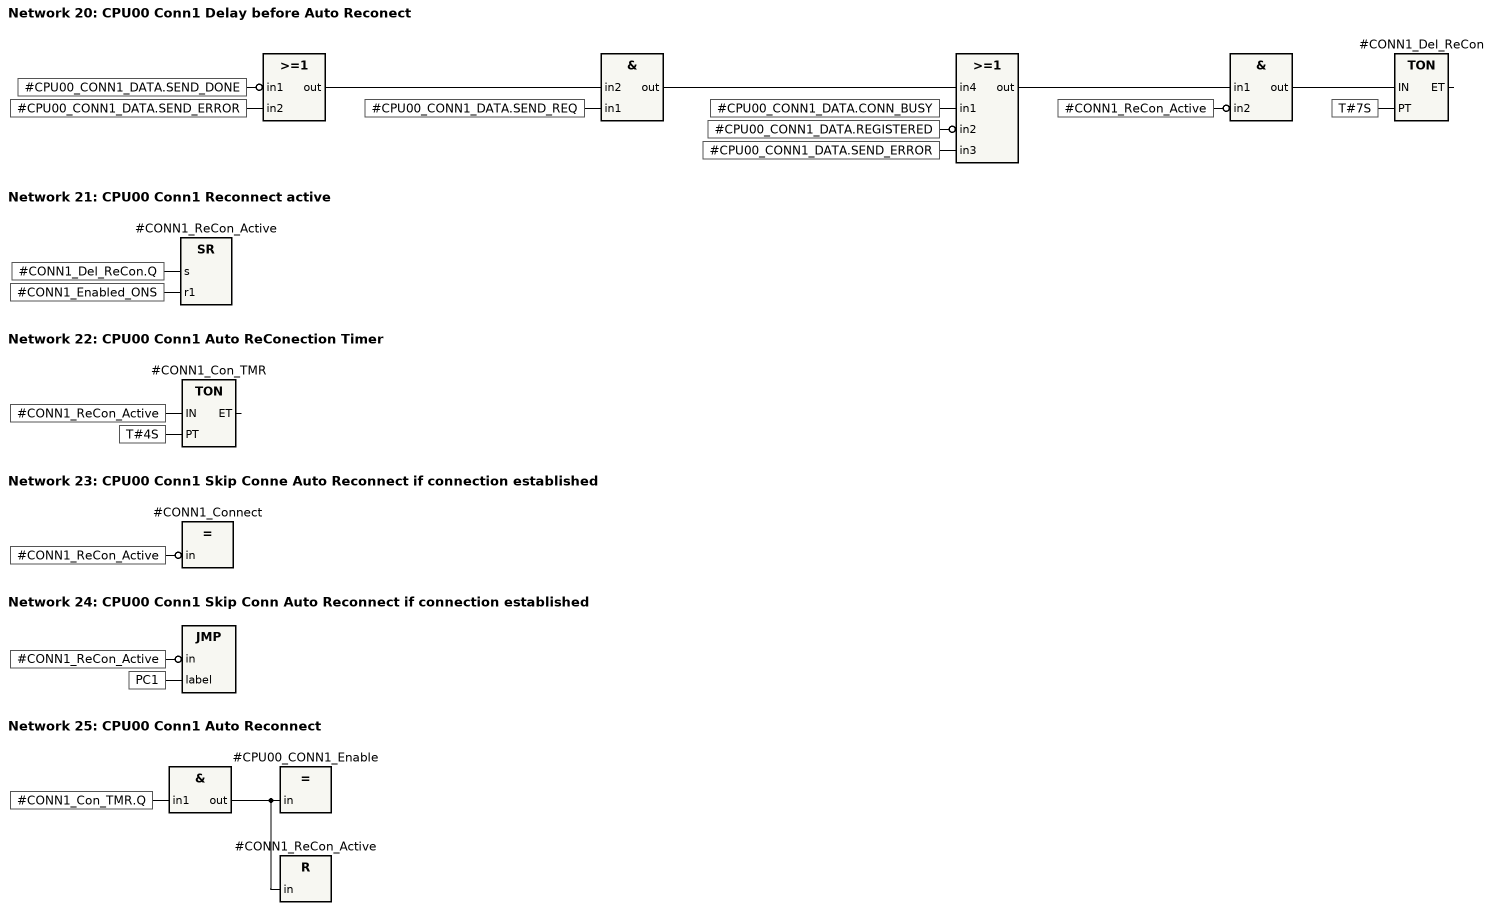
   #CONN1_Del_ReCon(IN := (((NOT #CPU00_CONN1_DATA.SEND_DONE OR #CPU00_CONN1_DATA.SEND_ERROR) AND #CPU00_CONN1_DATA.SEND_REQ) OR #CPU00_CONN1_DATA.CONN_BUSY OR NOT #CPU00_CONN1_DATA.REGISTERED OR #CPU00_CONN1_DATA.SEND_ERROR) AND NOT #CONN1_ReCon_Active,   // TON
                    PT := T#7S);
END_REGION

REGION Network 21: CPU00 Conn1 Reconnect active
   IF #CONN1_Del_ReCon.Q THEN
       #CONN1_ReCon_Active := TRUE;   // SR flip-flop
   END_IF;
   IF #CONN1_Enabled_ONS THEN #CONN1_ReCon_Active := FALSE; END_IF;
END_REGION

REGION Network 22: CPU00 Conn1 Auto ReConection Timer
   #CONN1_Con_TMR(IN := #CONN1_ReCon_Active, PT := T#4S);   // TON
END_REGION

REGION Network 23: CPU00 Conn1 Skip Conne Auto Reconnect if connection established
   #CONN1_Connect := NOT #CONN1_ReCon_Active;
END_REGION

REGION Network 24: CPU00 Conn1 Skip Conn Auto Reconnect if connection established
   IF NOT #CONN1_ReCon_Active THEN GOTO PC1; END_IF;
END_REGION

REGION Network 25: CPU00 Conn1 Auto Reconnect
   #CPU00_CONN1_Enable := #CONN1_Con_TMR.Q;
   IF #CONN1_Con_TMR.Q THEN #CONN1_ReCon_Active := FALSE; END_IF;
END_REGION

REGION Network 26 (STL): CPU00 Conn1 Set initial connection bit
   PC1:  O     #MASTER_LINK.FIRST_SCAN;
         O(;
         A     #CPU00_CONN1_Enable;
         FP    #CONN1_En_ONS;
         =     #CONN1_Enabled_ONS;
         A     #CONN1_Enabled_ONS;
         );
         =     #CONN1_INIT_COM;
END_REGION

REGION Network 27: CPU00 Conn1 Clear Bits to start initial conn and communication
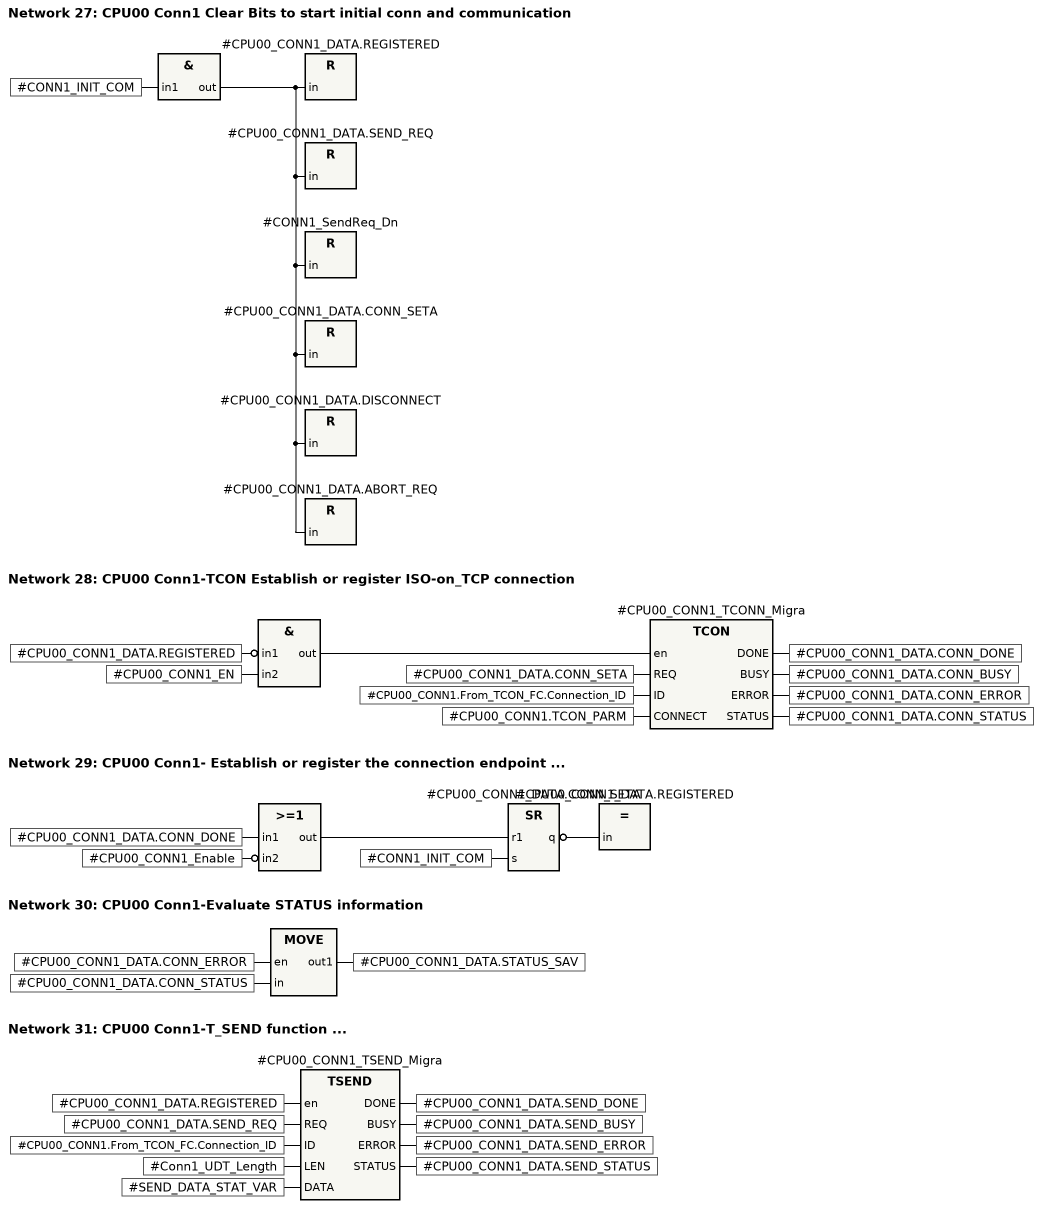
   IF #CONN1_INIT_COM THEN
       #CPU00_CONN1_DATA.REGISTERED := FALSE;
       #CPU00_CONN1_DATA.SEND_REQ := FALSE;
       #CONN1_SendReq_Dn := FALSE;
       #CPU00_CONN1_DATA.CONN_SETA := FALSE;
       #CPU00_CONN1_DATA.DISCONNECT := FALSE;
       #CPU00_CONN1_DATA.ABORT_REQ := FALSE;
   END_IF;
END_REGION

REGION Network 28: CPU00 Conn1-TCON Establish or register ISO-on_TCP connection
   // After the connection has been established, it is automatically monitored and 
   // maintained by the operating system of the CPU.
   // 
   // If the connection has been interrupted, by any line break or due to the remote 
   // communications partner, the active partner attempts to reestablish the 
   // connection.
   // 
   // Therefore, the FB 65 "TCON" may not be called again!
   IF NOT #CPU00_CONN1_DATA.REGISTERED AND #CPU00_CONN1_EN THEN
       #CPU00_CONN1_TCONN_Migra(REQ := #CPU00_CONN1_DATA.CONN_SETA,   // TCON
                               ID := #CPU00_CONN1.From_TCON_FC.Connection_ID,
                               CONNECT := #CPU00_CONN1.TCON_PARM,
                               DONE => #CPU00_CONN1_DATA.CONN_DONE,
                               BUSY => #CPU00_CONN1_DATA.CONN_BUSY,
                               ERROR => #CPU00_CONN1_DATA.CONN_ERROR,
                               STATUS => #CPU00_CONN1_DATA.CONN_STATUS);
   END_IF;
END_REGION

REGION Network 29: CPU00 Conn1- Establish or register the connection endpoint ...
   // while startup phase (initial).
   // 
   // Indication of the connection status:
   // 
   // a) If the CPU may establish the specified connection after Stop/Run  
   // immediately, the variable "REGISTERED" indicates HIGH (=1).
   // 
   // b) If the CPU is not able to establish the specified connection after Stop/Run, 
   // the variable "REGISTERED" remains LOW(=0).
   // 
   // c) Note: If the instance DB is loaded by the user, the variable "REGISTERED" 
   // indicates HIGH, although the connection may not be established yet. 
   // However, the FB64 "TRCV" would indicate the STATUS=0x80C4, as long as the 
   // connection has not been established.
   IF #CONN1_INIT_COM THEN
       #CPU00_CONN1_DATA.CONN_SETA := TRUE;   // SR flip-flop
   END_IF;
   IF #CPU00_CONN1_DATA.CONN_DONE OR NOT #CPU00_CONN1_Enable THEN
       #CPU00_CONN1_DATA.CONN_SETA := FALSE;
   END_IF;
   #CPU00_CONN1_DATA.REGISTERED := NOT #CPU00_CONN1_DATA.CONN_SETA;
END_REGION

REGION Network 30: CPU00 Conn1-Evaluate STATUS information
   // If ERROR occured then save STATUS!
   IF #CPU00_CONN1_DATA.CONN_ERROR THEN
       #CPU00_CONN1_DATA.STATUS_SAV := #CPU00_CONN1_DATA.CONN_STATUS;
   END_IF;
END_REGION

REGION Network 31: CPU00 Conn1-T_SEND function ...
   // if connection is established to transmit the data to the partner as a message.
   IF #CPU00_CONN1_DATA.REGISTERED THEN
       #CPU00_CONN1_TSEND_Migra(REQ := #CPU00_CONN1_DATA.SEND_REQ,   // TSEND
                               ID := #CPU00_CONN1.From_TCON_FC.Connection_ID,
                               LEN := #Conn1_UDT_Length,
                               DATA := #SEND_DATA_STAT_VAR,
                               DONE => #CPU00_CONN1_DATA.SEND_DONE,
                               BUSY => #CPU00_CONN1_DATA.SEND_BUSY,
                               ERROR => #CPU00_CONN1_DATA.SEND_ERROR,
                               STATUS => #CPU00_CONN1_DATA.SEND_STATUS);
   END_IF;
END_REGION

REGION Network 32: CPU00 Conn1-Generate the rising edge SEND_REQ to start T_SEND
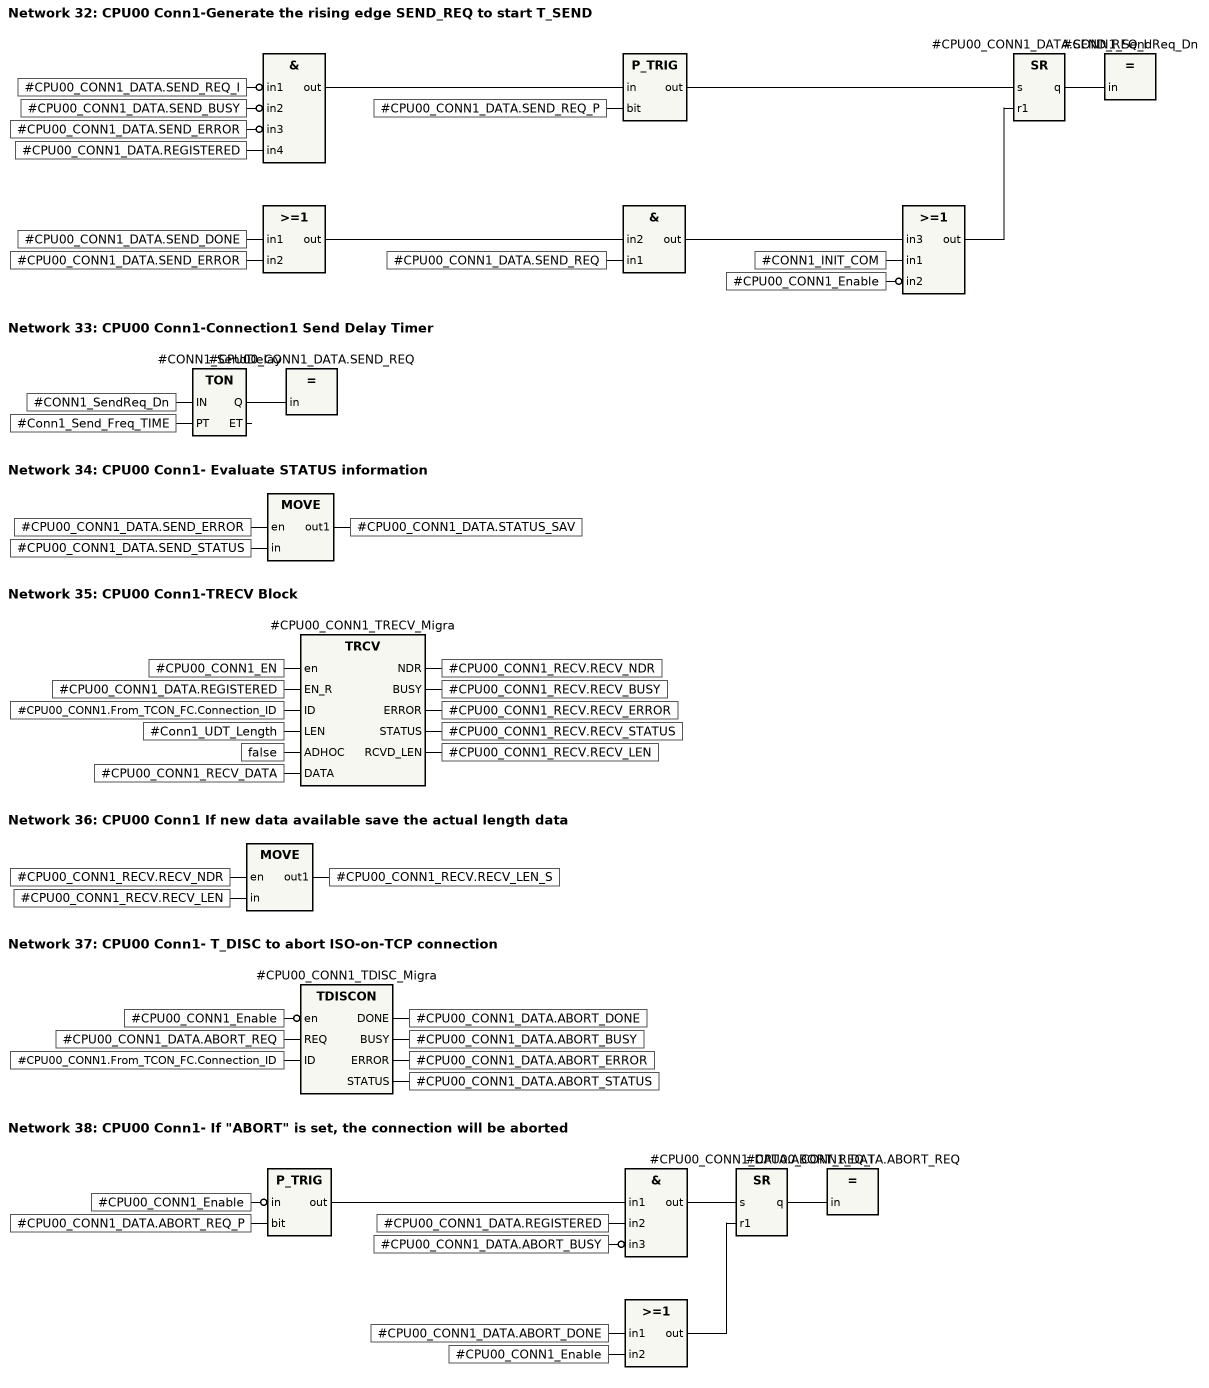
   #_w1 := NOT #CPU00_CONN1_DATA.SEND_REQ_I AND NOT #CPU00_CONN1_DATA.SEND_BUSY AND NOT #CPU00_CONN1_DATA.SEND_ERROR AND #CPU00_CONN1_DATA.REGISTERED;
   #_w2 := #_w1 AND NOT #CPU00_CONN1_DATA.SEND_REQ_P;   // rising edge
   #CPU00_CONN1_DATA.SEND_REQ_P := #_w1;
   IF #_w2 THEN
       #CPU00_CONN1_DATA.SEND_REQ_I := TRUE;   // SR flip-flop
   END_IF;
   IF ((#CPU00_CONN1_DATA.SEND_DONE OR #CPU00_CONN1_DATA.SEND_ERROR) AND #CPU00_CONN1_DATA.SEND_REQ) OR #CONN1_INIT_COM OR NOT #CPU00_CONN1_Enable THEN
       #CPU00_CONN1_DATA.SEND_REQ_I := FALSE;
   END_IF;
   #CONN1_SendReq_Dn := #CPU00_CONN1_DATA.SEND_REQ_I;
END_REGION

REGION Network 33: CPU00 Conn1-Connection1 Send Delay Timer
   #CONN1_SendDelay(IN := #CONN1_SendReq_Dn, PT := #Conn1_Send_Freq_TIME);   // TON
   #CPU00_CONN1_DATA.SEND_REQ := #CONN1_SendDelay.Q;
END_REGION

REGION Network 34: CPU00 Conn1- Evaluate STATUS information
   // If ERROR occured then save STATUS!
   IF #CPU00_CONN1_DATA.SEND_ERROR THEN
       #CPU00_CONN1_DATA.STATUS_SAV := #CPU00_CONN1_DATA.SEND_STATUS;
   END_IF;
END_REGION

REGION Network 35: CPU00 Conn1-TRECV Block
   IF #CPU00_CONN1_EN THEN
       #CPU00_CONN1_TRECV_Migra(EN_R := #CPU00_CONN1_DATA.REGISTERED,   // TRCV
                               ID := #CPU00_CONN1.From_TCON_FC.Connection_ID,
                               LEN := #Conn1_UDT_Length,
                               ADHOC := false,
                               DATA := #CPU00_CONN1_RECV_DATA,
                               NDR => #CPU00_CONN1_RECV.RECV_NDR,
                               BUSY => #CPU00_CONN1_RECV.RECV_BUSY,
                               ERROR => #CPU00_CONN1_RECV.RECV_ERROR,
                               STATUS => #CPU00_CONN1_RECV.RECV_STATUS,
                               RCVD_LEN => #CPU00_CONN1_RECV.RECV_LEN);
   END_IF;
END_REGION

REGION Network 36: CPU00 Conn1 If new data available save the actual length data
   IF #CPU00_CONN1_RECV.RECV_NDR THEN #CPU00_CONN1_RECV.RECV_LEN_S := #CPU00_CONN1_RECV.RECV_LEN; END_IF;
END_REGION

REGION Network 37: CPU00 Conn1- T_DISC to abort ISO-on-TCP connection
   // The FB 66 "TDISCON" terminates a communications connection from the CPU to a
   // communications partner.
   // 
   // An existing connection is terminated when FB 66 "TDISCON" is called or when the
   // CPU has gone into STOP mode. To reestablish the connection, the FB 65 "TCON" 
   // has to be invoked again.
   IF NOT #CPU00_CONN1_Enable THEN
       #CPU00_CONN1_TDISC_Migra(REQ := #CPU00_CONN1_DATA.ABORT_REQ,   // TDISCON
                               ID := #CPU00_CONN1.From_TCON_FC.Connection_ID,
                               DONE => #CPU00_CONN1_DATA.ABORT_DONE,
                               BUSY => #CPU00_CONN1_DATA.ABORT_BUSY,
                               ERROR => #CPU00_CONN1_DATA.ABORT_ERROR,
                               STATUS => #CPU00_CONN1_DATA.ABORT_STATUS);
   END_IF;
END_REGION

REGION Network 38: CPU00 Conn1- If "ABORT" is set, the connection will be aborted
   #_w1 := NOT #CPU00_CONN1_Enable AND NOT #CPU00_CONN1_DATA.ABORT_REQ_P;   // rising edge
   #CPU00_CONN1_DATA.ABORT_REQ_P := NOT #CPU00_CONN1_Enable;
   IF #_w1 AND #CPU00_CONN1_DATA.REGISTERED AND NOT #CPU00_CONN1_DATA.ABORT_BUSY THEN
       #CPU00_CONN1_DATA.ABORT_REQ_I := TRUE;   // SR flip-flop
   END_IF;
   IF #CPU00_CONN1_DATA.ABORT_DONE OR #CPU00_CONN1_Enable THEN
       #CPU00_CONN1_DATA.ABORT_REQ_I := FALSE;
   END_IF;
   #CPU00_CONN1_DATA.ABORT_REQ := #CPU00_CONN1_DATA.ABORT_REQ_I;
END_REGION

REGION Network 39: CPU00 Conn1-Communication OK
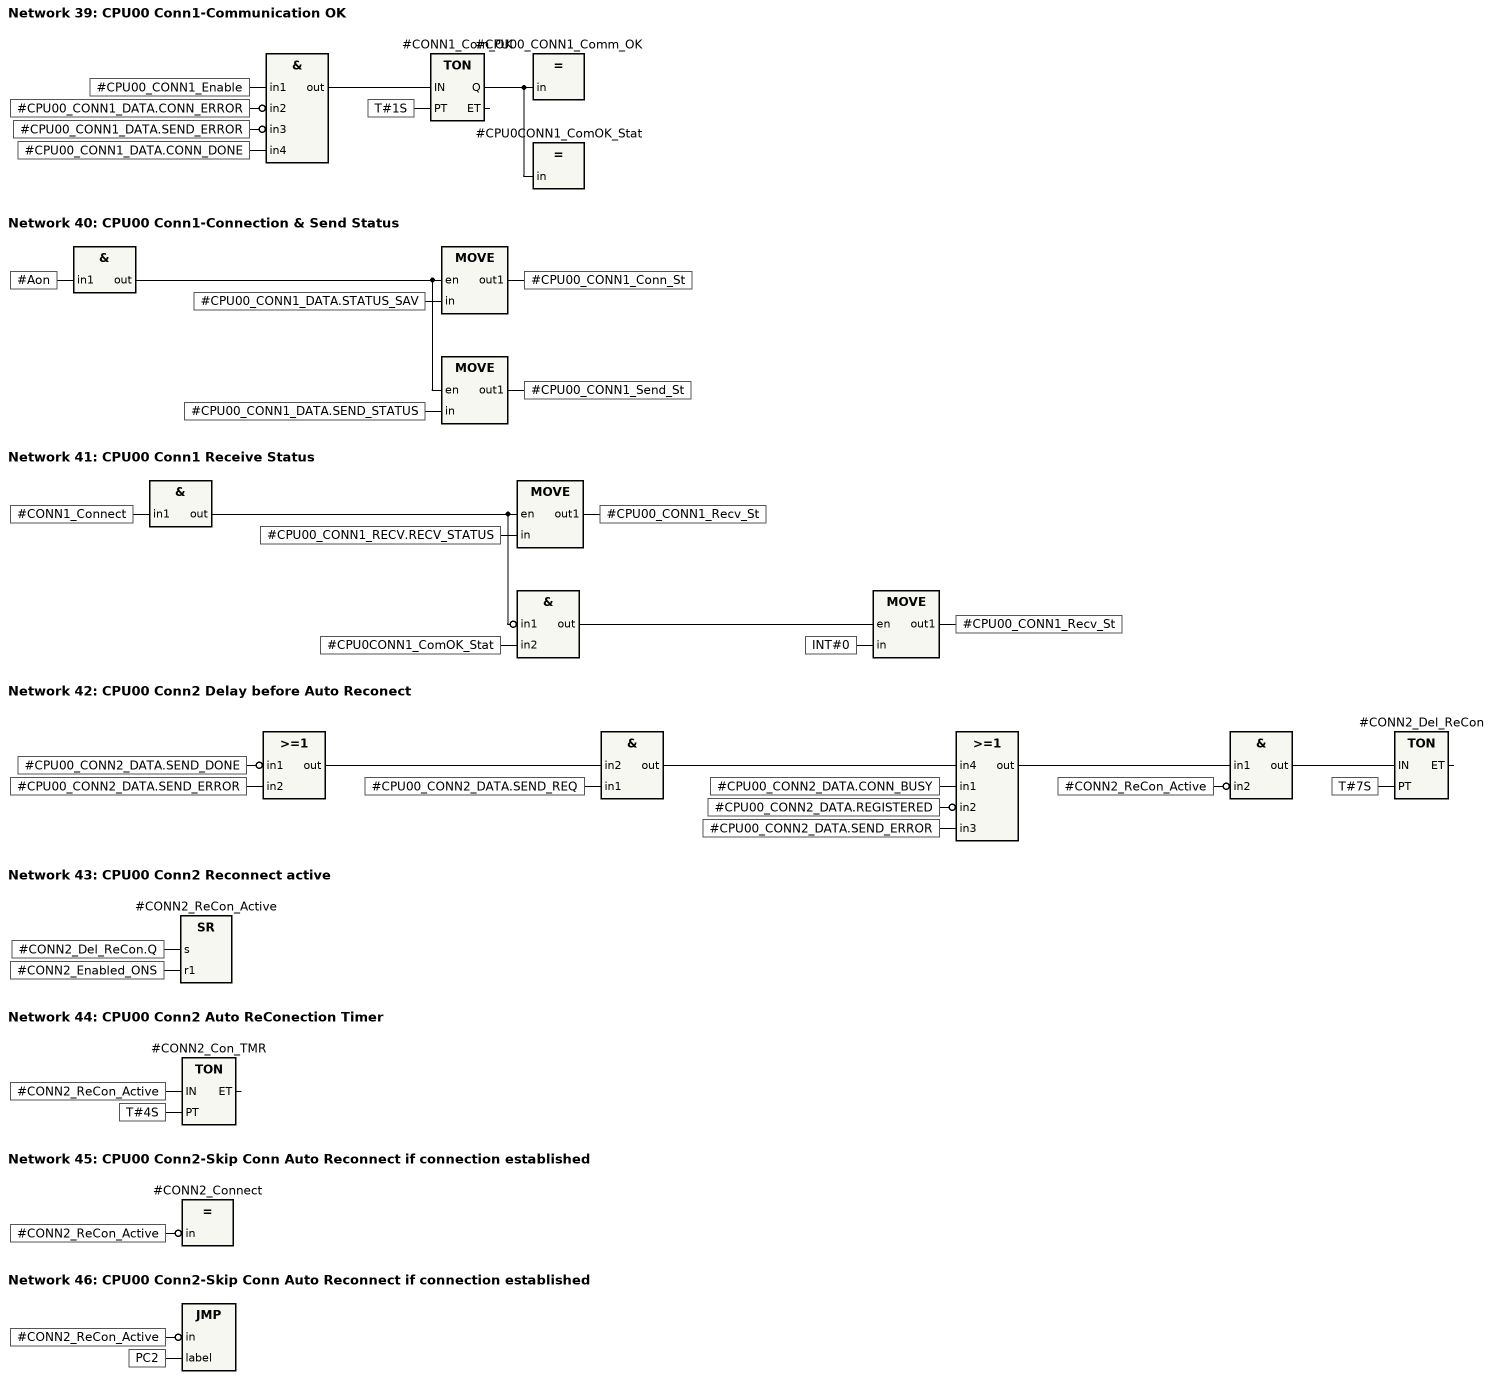
   #CONN1_Com_OK(IN := #CPU00_CONN1_Enable AND NOT #CPU00_CONN1_DATA.CONN_ERROR AND NOT #CPU00_CONN1_DATA.SEND_ERROR AND #CPU00_CONN1_DATA.CONN_DONE,   // TON
                 PT := T#1S);
   #CPU00_CONN1_Comm_OK := #CONN1_Com_OK.Q;
   #CPU0CONN1_ComOK_Stat := #CONN1_Com_OK.Q;
END_REGION

REGION Network 40: CPU00 Conn1-Connection & Send Status
   IF #Aon THEN
       #CPU00_CONN1_Conn_St := #CPU00_CONN1_DATA.STATUS_SAV;
       #CPU00_CONN1_Send_St := #CPU00_CONN1_DATA.SEND_STATUS;
   END_IF;
END_REGION

REGION Network 41: CPU00 Conn1 Receive Status
   IF #CONN1_Connect THEN #CPU00_CONN1_Recv_St := #CPU00_CONN1_RECV.RECV_STATUS; END_IF;
   IF NOT #CONN1_Connect AND #CPU0CONN1_ComOK_Stat THEN #CPU00_CONN1_Recv_St := INT#0; END_IF;
END_REGION

REGION Network 42: CPU00 Conn2 Delay before Auto Reconect
   #CONN2_Del_ReCon(IN := (((NOT #CPU00_CONN2_DATA.SEND_DONE OR #CPU00_CONN2_DATA.SEND_ERROR) AND #CPU00_CONN2_DATA.SEND_REQ) OR #CPU00_CONN2_DATA.CONN_BUSY OR NOT #CPU00_CONN2_DATA.REGISTERED OR #CPU00_CONN2_DATA.SEND_ERROR) AND NOT #CONN2_ReCon_Active,   // TON
                    PT := T#7S);
END_REGION

REGION Network 43: CPU00 Conn2 Reconnect active
   IF #CONN2_Del_ReCon.Q THEN
       #CONN2_ReCon_Active := TRUE;   // SR flip-flop
   END_IF;
   IF #CONN2_Enabled_ONS THEN #CONN2_ReCon_Active := FALSE; END_IF;
END_REGION

REGION Network 44: CPU00 Conn2 Auto ReConection Timer
   #CONN2_Con_TMR(IN := #CONN2_ReCon_Active, PT := T#4S);   // TON
END_REGION

REGION Network 45: CPU00 Conn2-Skip Conn Auto Reconnect if connection established
   #CONN2_Connect := NOT #CONN2_ReCon_Active;
END_REGION

REGION Network 46: CPU00 Conn2-Skip Conn Auto Reconnect if connection established
   IF NOT #CONN2_ReCon_Active THEN GOTO PC2; END_IF;
END_REGION

REGION Network 47: CPU00 Conn2 Auto Reconnect
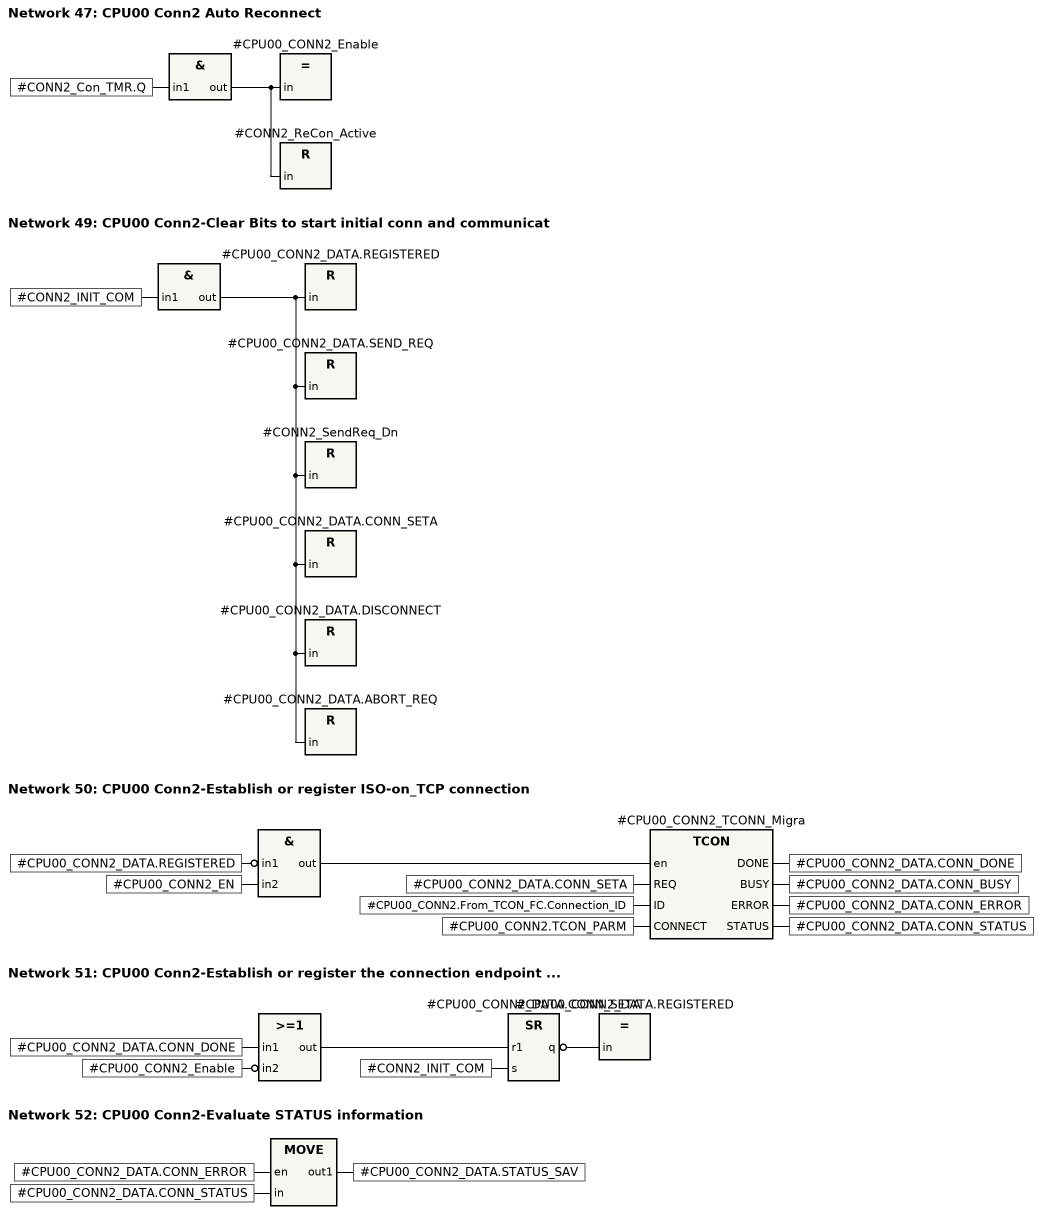
   #CPU00_CONN2_Enable := #CONN2_Con_TMR.Q;
   IF #CONN2_Con_TMR.Q THEN #CONN2_ReCon_Active := FALSE; END_IF;
END_REGION

REGION Network 48 (STL): CPU00 Conn2-Set initial connection bit - Connection 2 Link
   PC2:  O     #MASTER_LINK.FIRST_SCAN;
         O(;
         A     #CPU00_CONN2_Enable;
         FP    #CONN2_En_ONS;
         =     #CONN2_Enabled_ONS;
         A     #CONN2_Enabled_ONS;
         );
         =     #CONN2_INIT_COM;
END_REGION

REGION Network 49: CPU00 Conn2-Clear Bits to start initial conn and communicat
   IF #CONN2_INIT_COM THEN
       #CPU00_CONN2_DATA.REGISTERED := FALSE;
       #CPU00_CONN2_DATA.SEND_REQ := FALSE;
       #CONN2_SendReq_Dn := FALSE;
       #CPU00_CONN2_DATA.CONN_SETA := FALSE;
       #CPU00_CONN2_DATA.DISCONNECT := FALSE;
       #CPU00_CONN2_DATA.ABORT_REQ := FALSE;
   END_IF;
END_REGION

REGION Network 50: CPU00 Conn2-Establish or register ISO-on_TCP connection
   // After the connection has been established, it is automatically monitored and 
   // maintained by the operating system of the CPU.
   // 
   // If the connection has been interrupted, by any line break or due to the remote 
   // communications partner, the active partner attempts to reestablish the 
   // connection.
   // 
   // Therefore, the FB 65 "TCON" may not be called again!
   IF NOT #CPU00_CONN2_DATA.REGISTERED AND #CPU00_CONN2_EN THEN
       #CPU00_CONN2_TCONN_Migra(REQ := #CPU00_CONN2_DATA.CONN_SETA,   // TCON
                               ID := #CPU00_CONN2.From_TCON_FC.Connection_ID,
                               CONNECT := #CPU00_CONN2.TCON_PARM,
                               DONE => #CPU00_CONN2_DATA.CONN_DONE,
                               BUSY => #CPU00_CONN2_DATA.CONN_BUSY,
                               ERROR => #CPU00_CONN2_DATA.CONN_ERROR,
                               STATUS => #CPU00_CONN2_DATA.CONN_STATUS);
   END_IF;
END_REGION

REGION Network 51: CPU00 Conn2-Establish or register the connection endpoint ...
   // while startup phase (initial).
   // 
   // Indication of the connection status:
   // 
   // a) If the CPU may establish the specified connection after Stop/Run  
   // immediately, the variable "REGISTERED" indicates HIGH (=1).
   // 
   // b) If the CPU is not able to establish the specified connection after Stop/Run, 
   // the variable "REGISTERED" remains LOW(=0).
   // 
   // c) Note: If the instance DB is loaded by the user, the variable "REGISTERED" 
   // indicates HIGH, although the connection may not be established yet. 
   // However, the FB64 "TRCV" would indicate the STATUS=0x80C4, as long as the 
   // connection has not been established.
   IF #CONN2_INIT_COM THEN
       #CPU00_CONN2_DATA.CONN_SETA := TRUE;   // SR flip-flop
   END_IF;
   IF #CPU00_CONN2_DATA.CONN_DONE OR NOT #CPU00_CONN2_Enable THEN
       #CPU00_CONN2_DATA.CONN_SETA := FALSE;
   END_IF;
   #CPU00_CONN2_DATA.REGISTERED := NOT #CPU00_CONN2_DATA.CONN_SETA;
END_REGION

REGION Network 52: CPU00 Conn2-Evaluate STATUS information
   // If ERROR occured then save STATUS!
   IF #CPU00_CONN2_DATA.CONN_ERROR THEN
       #CPU00_CONN2_DATA.STATUS_SAV := #CPU00_CONN2_DATA.CONN_STATUS;
   END_IF;
END_REGION

REGION Network 53: CPU00 Conn2 - T_SEND function ...
   // if connection is established to transmit the data to the partner as a message.
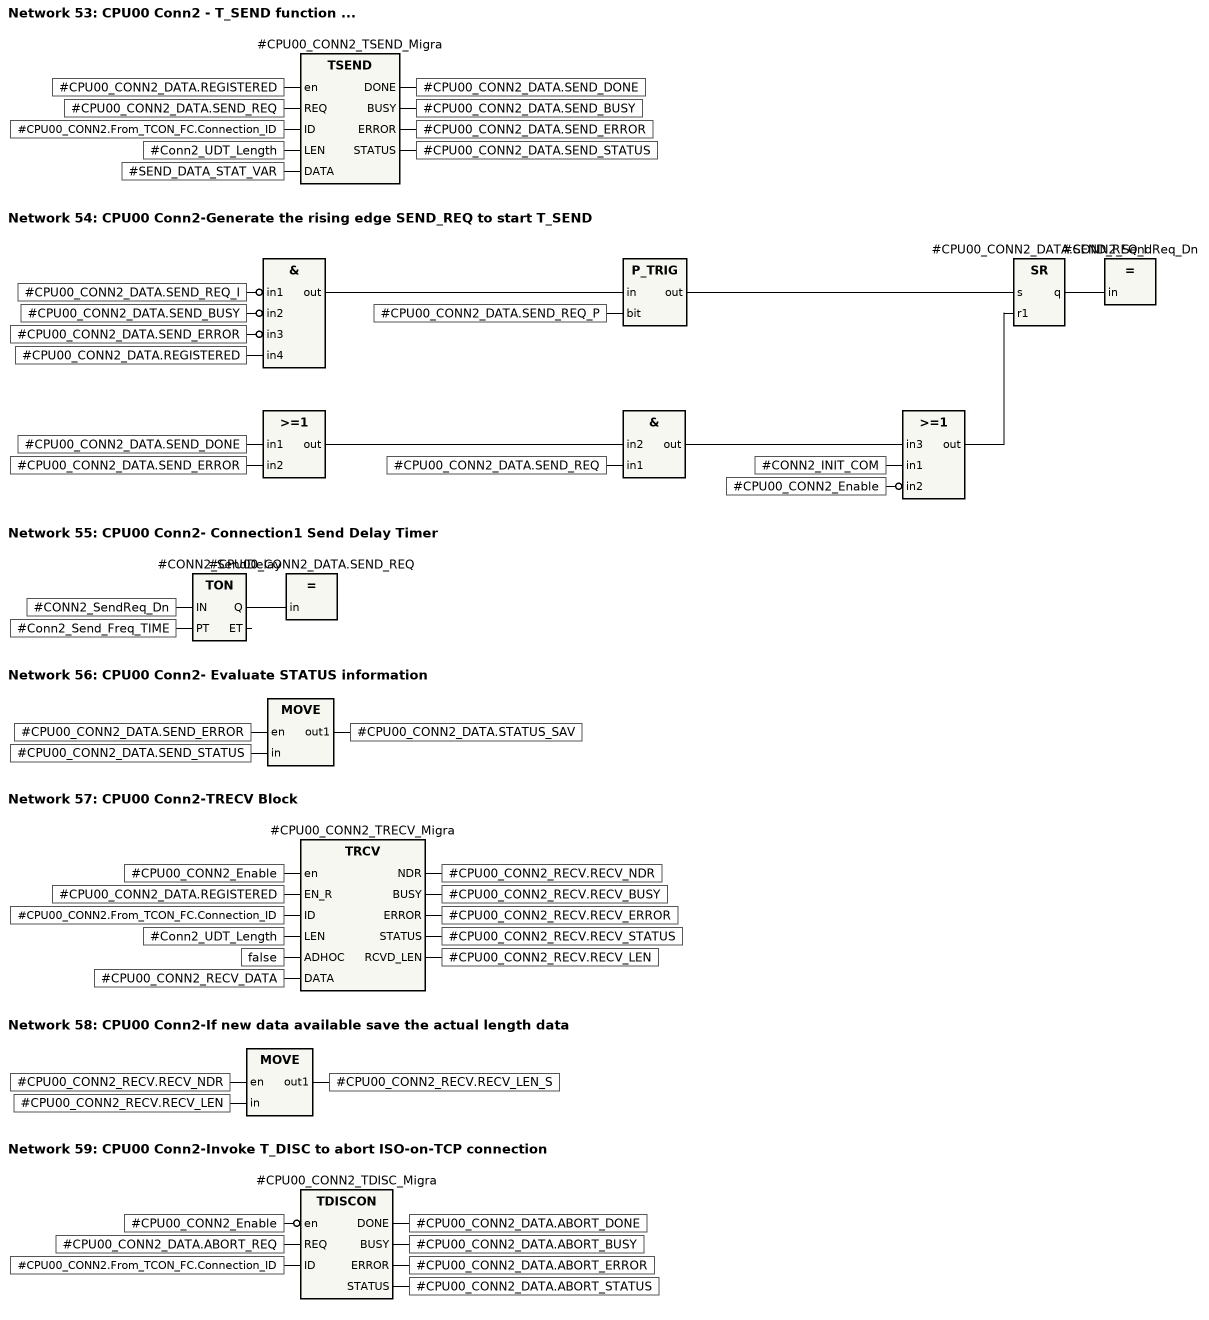
   IF #CPU00_CONN2_DATA.REGISTERED THEN
       #CPU00_CONN2_TSEND_Migra(REQ := #CPU00_CONN2_DATA.SEND_REQ,   // TSEND
                               ID := #CPU00_CONN2.From_TCON_FC.Connection_ID,
                               LEN := #Conn2_UDT_Length,
                               DATA := #SEND_DATA_STAT_VAR,
                               DONE => #CPU00_CONN2_DATA.SEND_DONE,
                               BUSY => #CPU00_CONN2_DATA.SEND_BUSY,
                               ERROR => #CPU00_CONN2_DATA.SEND_ERROR,
                               STATUS => #CPU00_CONN2_DATA.SEND_STATUS);
   END_IF;
END_REGION

REGION Network 54: CPU00 Conn2-Generate the rising edge SEND_REQ to start T_SEND
   #_w1 := NOT #CPU00_CONN2_DATA.SEND_REQ_I AND NOT #CPU00_CONN2_DATA.SEND_BUSY AND NOT #CPU00_CONN2_DATA.SEND_ERROR AND #CPU00_CONN2_DATA.REGISTERED;
   #_w2 := #_w1 AND NOT #CPU00_CONN2_DATA.SEND_REQ_P;   // rising edge
   #CPU00_CONN2_DATA.SEND_REQ_P := #_w1;
   IF #_w2 THEN
       #CPU00_CONN2_DATA.SEND_REQ_I := TRUE;   // SR flip-flop
   END_IF;
   IF ((#CPU00_CONN2_DATA.SEND_DONE OR #CPU00_CONN2_DATA.SEND_ERROR) AND #CPU00_CONN2_DATA.SEND_REQ) OR #CONN2_INIT_COM OR NOT #CPU00_CONN2_Enable THEN
       #CPU00_CONN2_DATA.SEND_REQ_I := FALSE;
   END_IF;
   #CONN2_SendReq_Dn := #CPU00_CONN2_DATA.SEND_REQ_I;
END_REGION

REGION Network 55: CPU00 Conn2- Connection1 Send Delay Timer
   #CONN2_SendDelay(IN := #CONN2_SendReq_Dn, PT := #Conn2_Send_Freq_TIME);   // TON
   #CPU00_CONN2_DATA.SEND_REQ := #CONN2_SendDelay.Q;
END_REGION

REGION Network 56: CPU00 Conn2- Evaluate STATUS information
   // If ERROR occured then save STATUS!
   IF #CPU00_CONN2_DATA.SEND_ERROR THEN
       #CPU00_CONN2_DATA.STATUS_SAV := #CPU00_CONN2_DATA.SEND_STATUS;
   END_IF;
END_REGION

REGION Network 57: CPU00 Conn2-TRECV Block
   IF #CPU00_CONN2_Enable THEN
       #CPU00_CONN2_TRECV_Migra(EN_R := #CPU00_CONN2_DATA.REGISTERED,   // TRCV
                               ID := #CPU00_CONN2.From_TCON_FC.Connection_ID,
                               LEN := #Conn2_UDT_Length,
                               ADHOC := false,
                               DATA := #CPU00_CONN2_RECV_DATA,
                               NDR => #CPU00_CONN2_RECV.RECV_NDR,
                               BUSY => #CPU00_CONN2_RECV.RECV_BUSY,
                               ERROR => #CPU00_CONN2_RECV.RECV_ERROR,
                               STATUS => #CPU00_CONN2_RECV.RECV_STATUS,
                               RCVD_LEN => #CPU00_CONN2_RECV.RECV_LEN);
   END_IF;
END_REGION

REGION Network 58: CPU00 Conn2-If new data available save the actual length data
   IF #CPU00_CONN2_RECV.RECV_NDR THEN #CPU00_CONN2_RECV.RECV_LEN_S := #CPU00_CONN2_RECV.RECV_LEN; END_IF;
END_REGION

REGION Network 59: CPU00 Conn2-Invoke T_DISC to abort ISO-on-TCP connection
   // The FB 66 "TDISCON" terminates a communications connection from the CPU to a
   // communications partner.
   // 
   // An existing connection is terminated when FB 66 "TDISCON" is called or when the
   // CPU has gone into STOP mode. To reestablish the connection, the FB 65 "TCON" 
   // has to be invoked again.
   IF NOT #CPU00_CONN2_Enable THEN
       #CPU00_CONN2_TDISC_Migra(REQ := #CPU00_CONN2_DATA.ABORT_REQ,   // TDISCON
                               ID := #CPU00_CONN2.From_TCON_FC.Connection_ID,
                               DONE => #CPU00_CONN2_DATA.ABORT_DONE,
                               BUSY => #CPU00_CONN2_DATA.ABORT_BUSY,
                               ERROR => #CPU00_CONN2_DATA.ABORT_ERROR,
                               STATUS => #CPU00_CONN2_DATA.ABORT_STATUS);
   END_IF;
END_REGION

REGION Network 60: CPU00 Conn2- If "ABORT" is set, the connection will be aborted
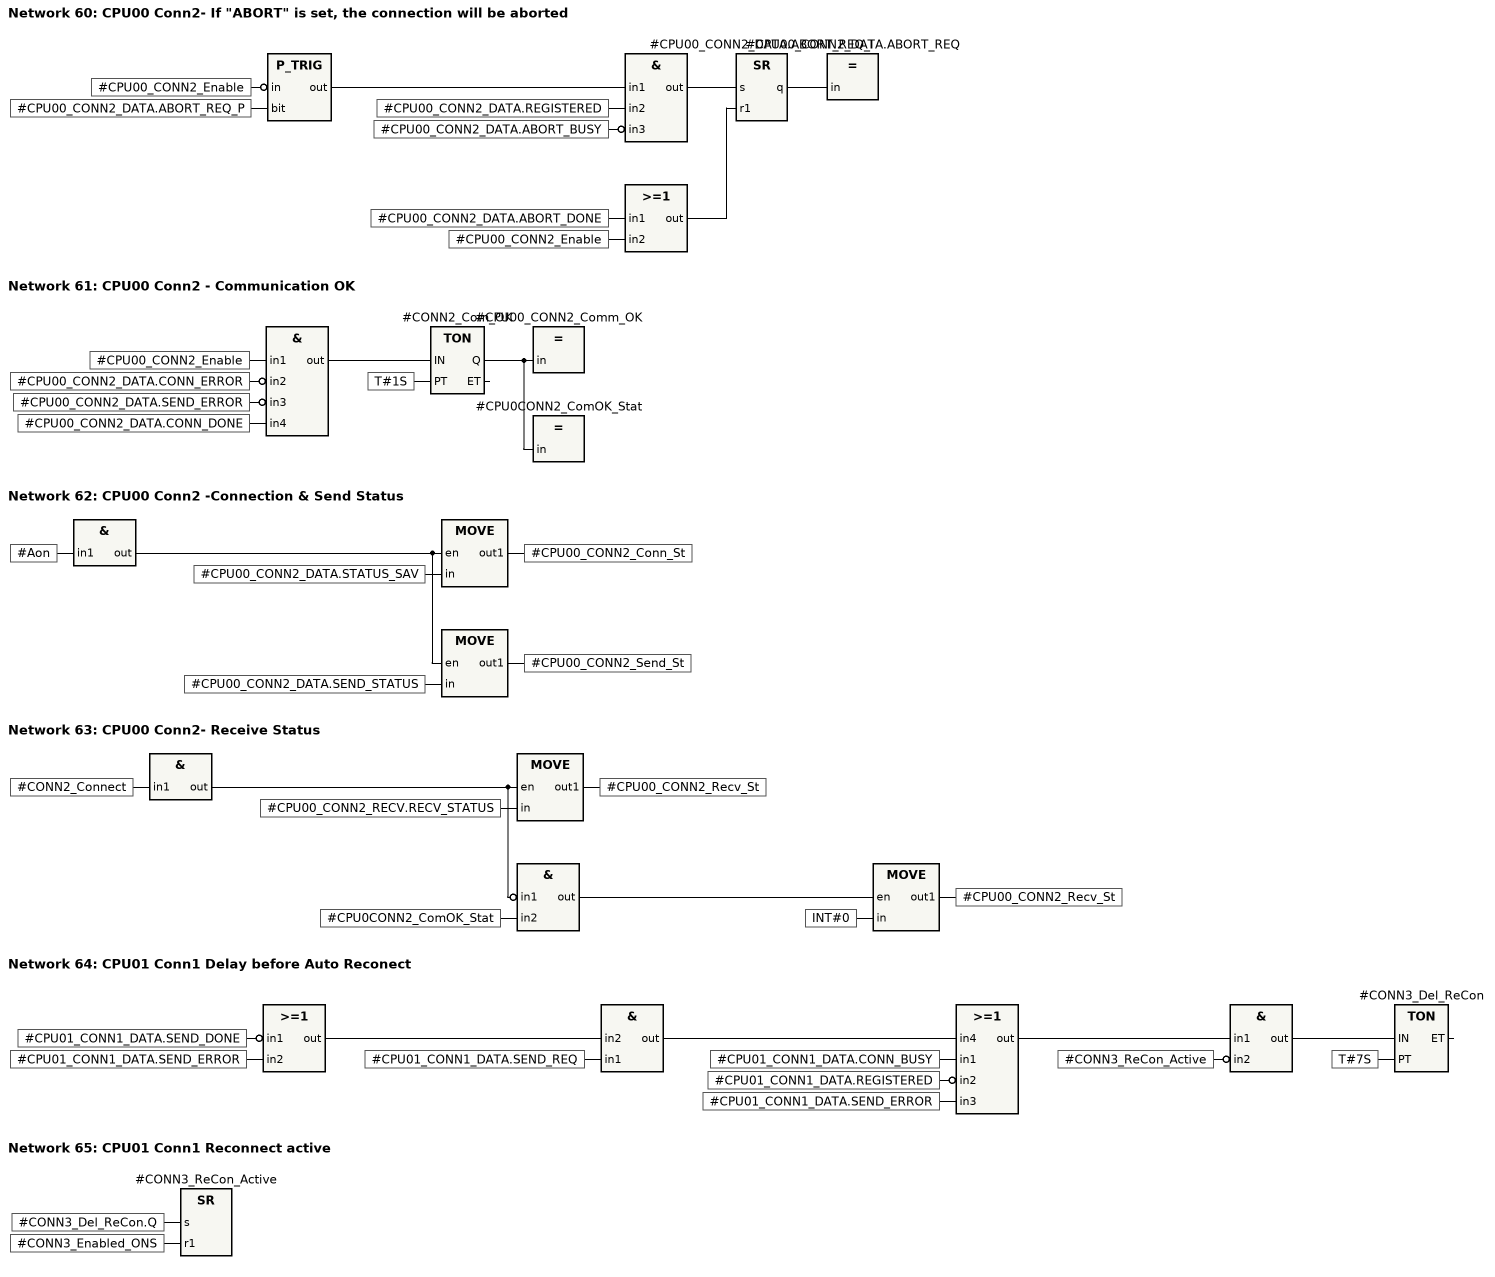
   #_w1 := NOT #CPU00_CONN2_Enable AND NOT #CPU00_CONN2_DATA.ABORT_REQ_P;   // rising edge
   #CPU00_CONN2_DATA.ABORT_REQ_P := NOT #CPU00_CONN2_Enable;
   IF #_w1 AND #CPU00_CONN2_DATA.REGISTERED AND NOT #CPU00_CONN2_DATA.ABORT_BUSY THEN
       #CPU00_CONN2_DATA.ABORT_REQ_I := TRUE;   // SR flip-flop
   END_IF;
   IF #CPU00_CONN2_DATA.ABORT_DONE OR #CPU00_CONN2_Enable THEN
       #CPU00_CONN2_DATA.ABORT_REQ_I := FALSE;
   END_IF;
   #CPU00_CONN2_DATA.ABORT_REQ := #CPU00_CONN2_DATA.ABORT_REQ_I;
END_REGION

REGION Network 61: CPU00 Conn2 - Communication OK
   #CONN2_Com_OK(IN := #CPU00_CONN2_Enable AND NOT #CPU00_CONN2_DATA.CONN_ERROR AND NOT #CPU00_CONN2_DATA.SEND_ERROR AND #CPU00_CONN2_DATA.CONN_DONE,   // TON
                 PT := T#1S);
   #CPU00_CONN2_Comm_OK := #CONN2_Com_OK.Q;
   #CPU0CONN2_ComOK_Stat := #CONN2_Com_OK.Q;
END_REGION

REGION Network 62: CPU00 Conn2 -Connection & Send Status
   IF #Aon THEN
       #CPU00_CONN2_Conn_St := #CPU00_CONN2_DATA.STATUS_SAV;
       #CPU00_CONN2_Send_St := #CPU00_CONN2_DATA.SEND_STATUS;
   END_IF;
END_REGION

REGION Network 63: CPU00 Conn2- Receive Status
   IF #CONN2_Connect THEN #CPU00_CONN2_Recv_St := #CPU00_CONN2_RECV.RECV_STATUS; END_IF;
   IF NOT #CONN2_Connect AND #CPU0CONN2_ComOK_Stat THEN #CPU00_CONN2_Recv_St := INT#0; END_IF;
END_REGION

REGION Network 64: CPU01 Conn1 Delay before Auto Reconect
   #CONN3_Del_ReCon(IN := (((NOT #CPU01_CONN1_DATA.SEND_DONE OR #CPU01_CONN1_DATA.SEND_ERROR) AND #CPU01_CONN1_DATA.SEND_REQ) OR #CPU01_CONN1_DATA.CONN_BUSY OR NOT #CPU01_CONN1_DATA.REGISTERED OR #CPU01_CONN1_DATA.SEND_ERROR) AND NOT #CONN3_ReCon_Active,   // TON
                    PT := T#7S);
END_REGION

REGION Network 65: CPU01 Conn1 Reconnect active
   IF #CONN3_Del_ReCon.Q THEN
       #CONN3_ReCon_Active := TRUE;   // SR flip-flop
   END_IF;
   IF #CONN3_Enabled_ONS THEN #CONN3_ReCon_Active := FALSE; END_IF;
END_REGION

REGION Network 66: CPU01 Conn1 Auto ReConection Timer
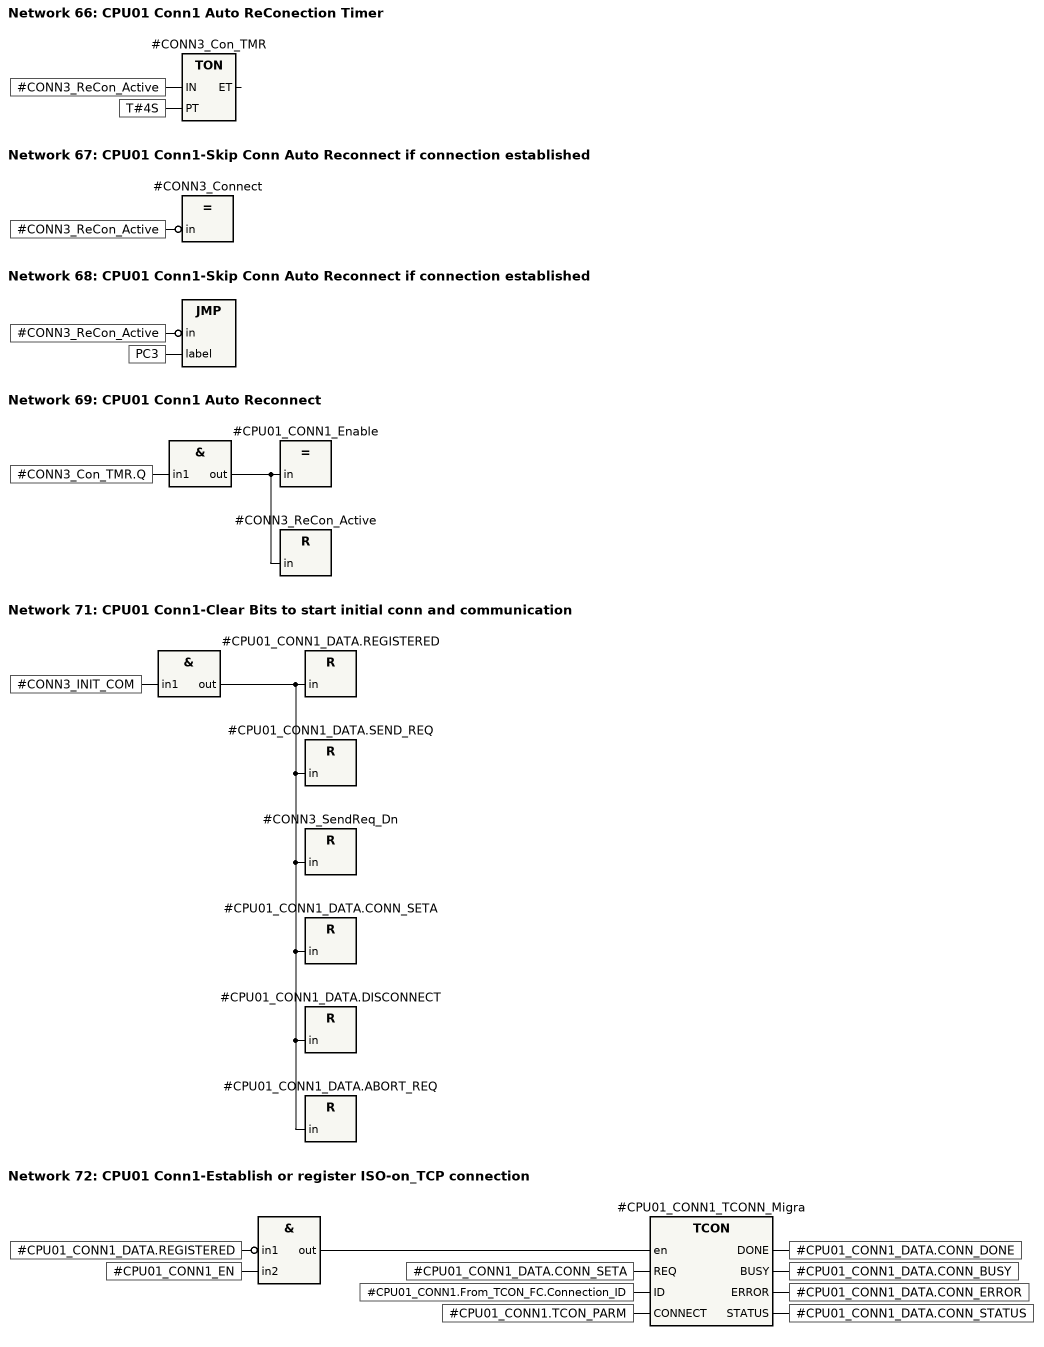
   #CONN3_Con_TMR(IN := #CONN3_ReCon_Active, PT := T#4S);   // TON
END_REGION

REGION Network 67: CPU01 Conn1-Skip Conn Auto Reconnect if connection established
   #CONN3_Connect := NOT #CONN3_ReCon_Active;
END_REGION

REGION Network 68: CPU01 Conn1-Skip Conn Auto Reconnect if connection established
   IF NOT #CONN3_ReCon_Active THEN GOTO PC3; END_IF;
END_REGION

REGION Network 69: CPU01 Conn1 Auto Reconnect
   #CPU01_CONN1_Enable := #CONN3_Con_TMR.Q;
   IF #CONN3_Con_TMR.Q THEN #CONN3_ReCon_Active := FALSE; END_IF;
END_REGION

REGION Network 70 (STL): CPU01 Conn1-Set initial connection bit - Connection 3 Link
   PC3:  O     #MASTER_LINK.FIRST_SCAN;
         O(;
         A     #CPU01_CONN1_Enable;
         FP    #CONN3_En_ONS;
         =     #CONN3_Enabled_ONS;
         A     #CONN3_Enabled_ONS;
         );
         =     #CONN3_INIT_COM;
END_REGION

REGION Network 71: CPU01 Conn1-Clear Bits to start initial conn and communication
   IF #CONN3_INIT_COM THEN
       #CPU01_CONN1_DATA.REGISTERED := FALSE;
       #CPU01_CONN1_DATA.SEND_REQ := FALSE;
       #CONN3_SendReq_Dn := FALSE;
       #CPU01_CONN1_DATA.CONN_SETA := FALSE;
       #CPU01_CONN1_DATA.DISCONNECT := FALSE;
       #CPU01_CONN1_DATA.ABORT_REQ := FALSE;
   END_IF;
END_REGION

REGION Network 72: CPU01 Conn1-Establish or register ISO-on_TCP connection
   // After the connection has been established, it is automatically monitored and 
   // maintained by the operating system of the CPU.
   // 
   // If the connection has been interrupted, by any line break or due to the remote 
   // communications partner, the active partner attempts to reestablish the 
   // connection.
   // 
   // Therefore, the FB 65 "TCON" may not be called again!
   IF NOT #CPU01_CONN1_DATA.REGISTERED AND #CPU01_CONN1_EN THEN
       #CPU01_CONN1_TCONN_Migra(REQ := #CPU01_CONN1_DATA.CONN_SETA,   // TCON
                               ID := #CPU01_CONN1.From_TCON_FC.Connection_ID,
                               CONNECT := #CPU01_CONN1.TCON_PARM,
                               DONE => #CPU01_CONN1_DATA.CONN_DONE,
                               BUSY => #CPU01_CONN1_DATA.CONN_BUSY,
                               ERROR => #CPU01_CONN1_DATA.CONN_ERROR,
                               STATUS => #CPU01_CONN1_DATA.CONN_STATUS);
   END_IF;
END_REGION

REGION Network 73: CPU01 Conn1-Establish or register the connection endpoint ...
   // while startup phase (initial).
   // 
   // Indication of the connection status:
   // 
   // a) If the CPU may establish the specified connection after Stop/Run  
   // immediately, the variable "REGISTERED" indicates HIGH (=1).
   // 
   // b) If the CPU is not able to establish the specified connection after Stop/Run, 
   // the variable "REGISTERED" remains LOW(=0).
   // 
   // c) Note: If the instance DB is loaded by the user, the variable "REGISTERED" 
   // indicates HIGH, although the connection may not be established yet. 
   // However, the FB64 "TRCV" would indicate the STATUS=0x80C4, as long as the 
   // connection has not been established.
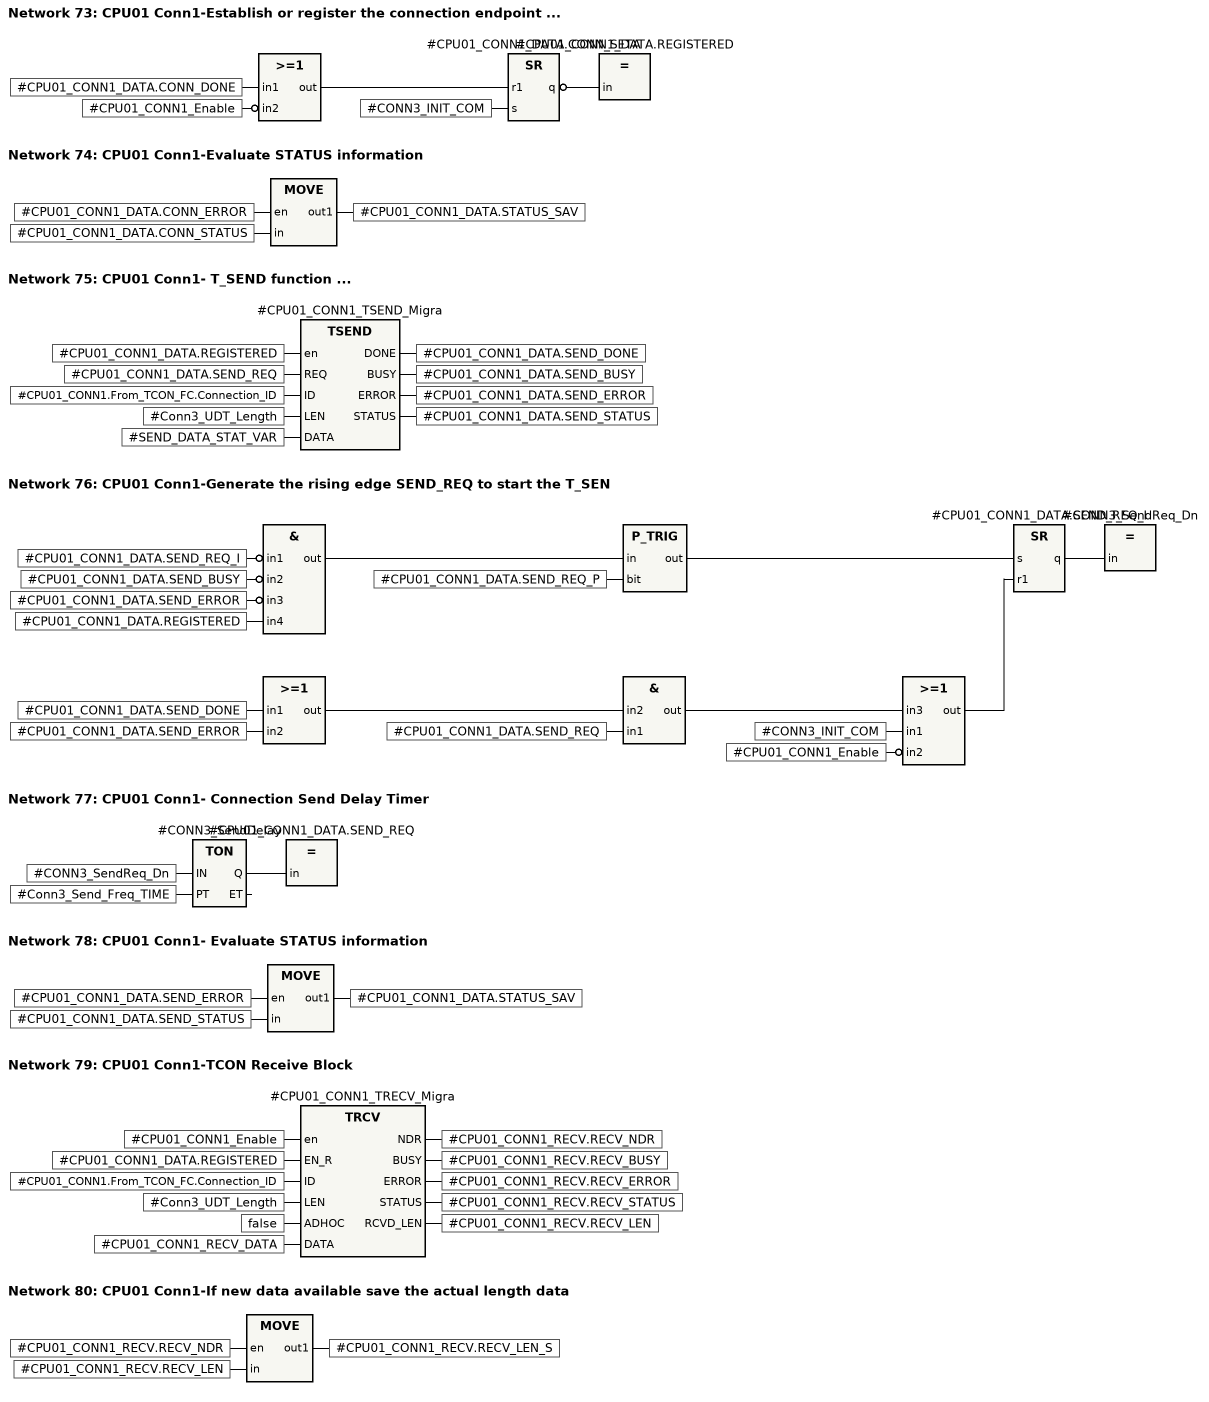
   IF #CONN3_INIT_COM THEN
       #CPU01_CONN1_DATA.CONN_SETA := TRUE;   // SR flip-flop
   END_IF;
   IF #CPU01_CONN1_DATA.CONN_DONE OR NOT #CPU01_CONN1_Enable THEN
       #CPU01_CONN1_DATA.CONN_SETA := FALSE;
   END_IF;
   #CPU01_CONN1_DATA.REGISTERED := NOT #CPU01_CONN1_DATA.CONN_SETA;
END_REGION

REGION Network 74: CPU01 Conn1-Evaluate STATUS information
   // If ERROR occured then save STATUS!
   IF #CPU01_CONN1_DATA.CONN_ERROR THEN
       #CPU01_CONN1_DATA.STATUS_SAV := #CPU01_CONN1_DATA.CONN_STATUS;
   END_IF;
END_REGION

REGION Network 75: CPU01 Conn1- T_SEND function ...
   // if connection is established to transmit the data to the partner as a message.
   IF #CPU01_CONN1_DATA.REGISTERED THEN
       #CPU01_CONN1_TSEND_Migra(REQ := #CPU01_CONN1_DATA.SEND_REQ,   // TSEND
                               ID := #CPU01_CONN1.From_TCON_FC.Connection_ID,
                               LEN := #Conn3_UDT_Length,
                               DATA := #SEND_DATA_STAT_VAR,
                               DONE => #CPU01_CONN1_DATA.SEND_DONE,
                               BUSY => #CPU01_CONN1_DATA.SEND_BUSY,
                               ERROR => #CPU01_CONN1_DATA.SEND_ERROR,
                               STATUS => #CPU01_CONN1_DATA.SEND_STATUS);
   END_IF;
END_REGION

REGION Network 76: CPU01 Conn1-Generate the rising edge SEND_REQ to start the T_SEN
   #_w1 := NOT #CPU01_CONN1_DATA.SEND_REQ_I AND NOT #CPU01_CONN1_DATA.SEND_BUSY AND NOT #CPU01_CONN1_DATA.SEND_ERROR AND #CPU01_CONN1_DATA.REGISTERED;
   #_w2 := #_w1 AND NOT #CPU01_CONN1_DATA.SEND_REQ_P;   // rising edge
   #CPU01_CONN1_DATA.SEND_REQ_P := #_w1;
   IF #_w2 THEN
       #CPU01_CONN1_DATA.SEND_REQ_I := TRUE;   // SR flip-flop
   END_IF;
   IF ((#CPU01_CONN1_DATA.SEND_DONE OR #CPU01_CONN1_DATA.SEND_ERROR) AND #CPU01_CONN1_DATA.SEND_REQ) OR #CONN3_INIT_COM OR NOT #CPU01_CONN1_Enable THEN
       #CPU01_CONN1_DATA.SEND_REQ_I := FALSE;
   END_IF;
   #CONN3_SendReq_Dn := #CPU01_CONN1_DATA.SEND_REQ_I;
END_REGION

REGION Network 77: CPU01 Conn1- Connection Send Delay Timer
   #CONN3_SendDelay(IN := #CONN3_SendReq_Dn, PT := #Conn3_Send_Freq_TIME);   // TON
   #CPU01_CONN1_DATA.SEND_REQ := #CONN3_SendDelay.Q;
END_REGION

REGION Network 78: CPU01 Conn1- Evaluate STATUS information
   // If ERROR occured then save STATUS!
   IF #CPU01_CONN1_DATA.SEND_ERROR THEN
       #CPU01_CONN1_DATA.STATUS_SAV := #CPU01_CONN1_DATA.SEND_STATUS;
   END_IF;
END_REGION

REGION Network 79: CPU01 Conn1-TCON Receive Block
   IF #CPU01_CONN1_Enable THEN
       #CPU01_CONN1_TRECV_Migra(EN_R := #CPU01_CONN1_DATA.REGISTERED,   // TRCV
                               ID := #CPU01_CONN1.From_TCON_FC.Connection_ID,
                               LEN := #Conn3_UDT_Length,
                               ADHOC := false,
                               DATA := #CPU01_CONN1_RECV_DATA,
                               NDR => #CPU01_CONN1_RECV.RECV_NDR,
                               BUSY => #CPU01_CONN1_RECV.RECV_BUSY,
                               ERROR => #CPU01_CONN1_RECV.RECV_ERROR,
                               STATUS => #CPU01_CONN1_RECV.RECV_STATUS,
                               RCVD_LEN => #CPU01_CONN1_RECV.RECV_LEN);
   END_IF;
END_REGION

REGION Network 80: CPU01 Conn1-If new data available save the actual length data
   IF #CPU01_CONN1_RECV.RECV_NDR THEN #CPU01_CONN1_RECV.RECV_LEN_S := #CPU01_CONN1_RECV.RECV_LEN; END_IF;
END_REGION

REGION Network 81: CPU01 Conn1-Invoke T_DISC to abort ISO-on-TCP connection
   // The FB 66 "TDISCON" terminates a communications connection from the CPU to a
   // communications partner.
   // 
   // An existing connection is terminated when FB 66 "TDISCON" is called or when the
   // CPU has gone into STOP mode. To reestablish the connection, the FB 65 "TCON" 
   // has to be invoked again.
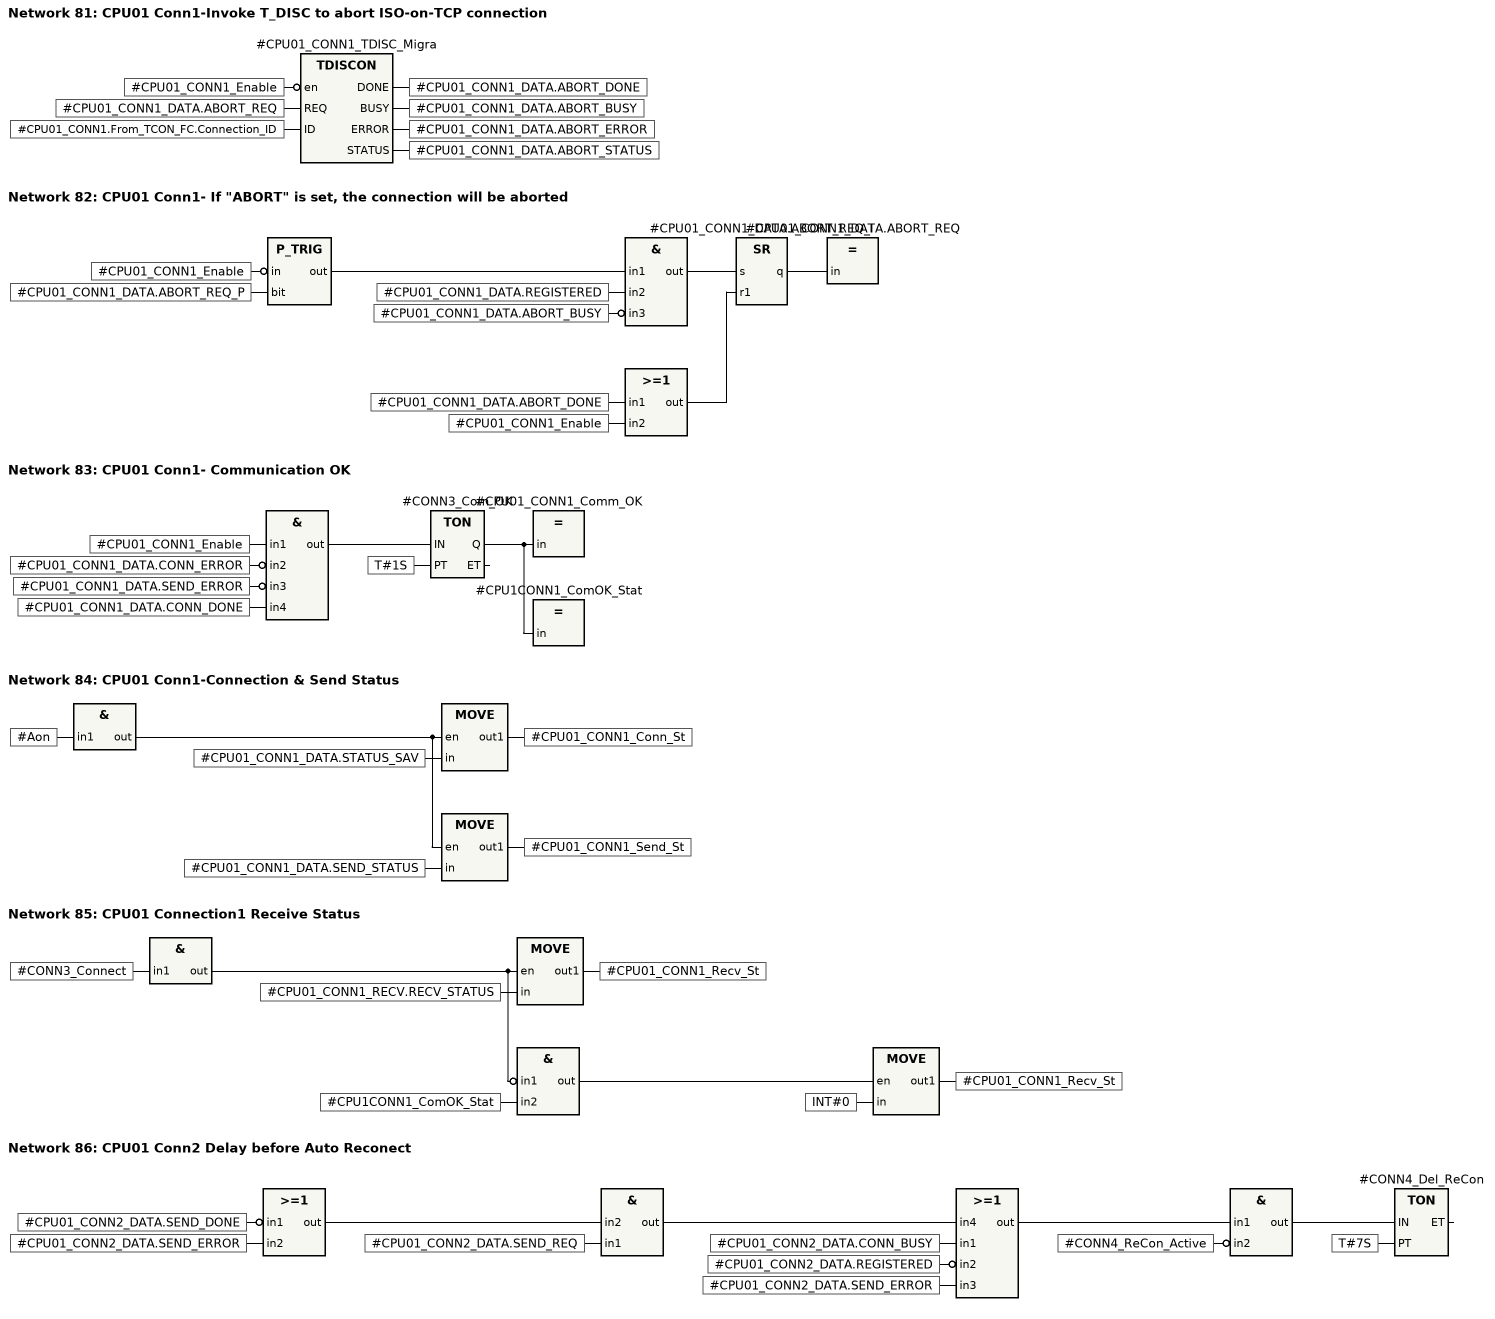
   IF NOT #CPU01_CONN1_Enable THEN
       #CPU01_CONN1_TDISC_Migra(REQ := #CPU01_CONN1_DATA.ABORT_REQ,   // TDISCON
                               ID := #CPU01_CONN1.From_TCON_FC.Connection_ID,
                               DONE => #CPU01_CONN1_DATA.ABORT_DONE,
                               BUSY => #CPU01_CONN1_DATA.ABORT_BUSY,
                               ERROR => #CPU01_CONN1_DATA.ABORT_ERROR,
                               STATUS => #CPU01_CONN1_DATA.ABORT_STATUS);
   END_IF;
END_REGION

REGION Network 82: CPU01 Conn1- If "ABORT" is set, the connection will be aborted
   #_w1 := NOT #CPU01_CONN1_Enable AND NOT #CPU01_CONN1_DATA.ABORT_REQ_P;   // rising edge
   #CPU01_CONN1_DATA.ABORT_REQ_P := NOT #CPU01_CONN1_Enable;
   IF #_w1 AND #CPU01_CONN1_DATA.REGISTERED AND NOT #CPU01_CONN1_DATA.ABORT_BUSY THEN
       #CPU01_CONN1_DATA.ABORT_REQ_I := TRUE;   // SR flip-flop
   END_IF;
   IF #CPU01_CONN1_DATA.ABORT_DONE OR #CPU01_CONN1_Enable THEN
       #CPU01_CONN1_DATA.ABORT_REQ_I := FALSE;
   END_IF;
   #CPU01_CONN1_DATA.ABORT_REQ := #CPU01_CONN1_DATA.ABORT_REQ_I;
END_REGION

REGION Network 83: CPU01 Conn1- Communication OK
   #CONN3_Com_OK(IN := #CPU01_CONN1_Enable AND NOT #CPU01_CONN1_DATA.CONN_ERROR AND NOT #CPU01_CONN1_DATA.SEND_ERROR AND #CPU01_CONN1_DATA.CONN_DONE,   // TON
                 PT := T#1S);
   #CPU01_CONN1_Comm_OK := #CONN3_Com_OK.Q;
   #CPU1CONN1_ComOK_Stat := #CONN3_Com_OK.Q;
END_REGION

REGION Network 84: CPU01 Conn1-Connection & Send Status
   IF #Aon THEN
       #CPU01_CONN1_Conn_St := #CPU01_CONN1_DATA.STATUS_SAV;
       #CPU01_CONN1_Send_St := #CPU01_CONN1_DATA.SEND_STATUS;
   END_IF;
END_REGION

REGION Network 85: CPU01 Connection1 Receive Status
   IF #CONN3_Connect THEN #CPU01_CONN1_Recv_St := #CPU01_CONN1_RECV.RECV_STATUS; END_IF;
   IF NOT #CONN3_Connect AND #CPU1CONN1_ComOK_Stat THEN #CPU01_CONN1_Recv_St := INT#0; END_IF;
END_REGION

REGION Network 86: CPU01 Conn2 Delay before Auto Reconect
   #CONN4_Del_ReCon(IN := (((NOT #CPU01_CONN2_DATA.SEND_DONE OR #CPU01_CONN2_DATA.SEND_ERROR) AND #CPU01_CONN2_DATA.SEND_REQ) OR #CPU01_CONN2_DATA.CONN_BUSY OR NOT #CPU01_CONN2_DATA.REGISTERED OR #CPU01_CONN2_DATA.SEND_ERROR) AND NOT #CONN4_ReCon_Active,   // TON
                    PT := T#7S);
END_REGION

REGION Network 87: CPU01 Conn2 Reconnect active
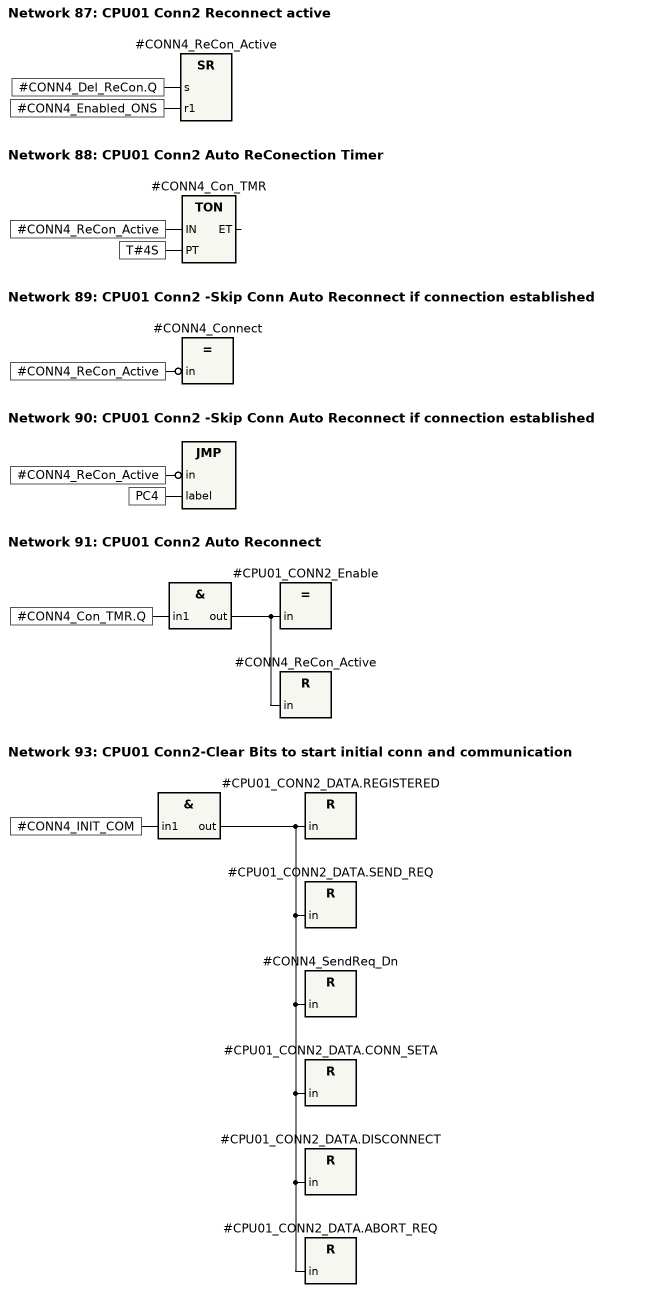
   IF #CONN4_Del_ReCon.Q THEN
       #CONN4_ReCon_Active := TRUE;   // SR flip-flop
   END_IF;
   IF #CONN4_Enabled_ONS THEN #CONN4_ReCon_Active := FALSE; END_IF;
END_REGION

REGION Network 88: CPU01 Conn2 Auto ReConection Timer
   #CONN4_Con_TMR(IN := #CONN4_ReCon_Active, PT := T#4S);   // TON
END_REGION

REGION Network 89: CPU01 Conn2 -Skip Conn Auto Reconnect if connection established
   #CONN4_Connect := NOT #CONN4_ReCon_Active;
END_REGION

REGION Network 90: CPU01 Conn2 -Skip Conn Auto Reconnect if connection established
   IF NOT #CONN4_ReCon_Active THEN GOTO PC4; END_IF;
END_REGION

REGION Network 91: CPU01 Conn2 Auto Reconnect
   #CPU01_CONN2_Enable := #CONN4_Con_TMR.Q;
   IF #CONN4_Con_TMR.Q THEN #CONN4_ReCon_Active := FALSE; END_IF;
END_REGION

REGION Network 92 (STL): CPU01 Conn2 Set initial connection bit
   PC4:  O     #MASTER_LINK.FIRST_SCAN;
         O(;
         A     #CPU01_CONN2_Enable;
         FP    #CONN4_En_ONS;
         =     #CONN4_Enabled_ONS;
         A     #CONN4_Enabled_ONS;
         );
         =     #CONN4_INIT_COM;
END_REGION

REGION Network 93: CPU01 Conn2-Clear Bits to start initial conn and communication
   IF #CONN4_INIT_COM THEN
       #CPU01_CONN2_DATA.REGISTERED := FALSE;
       #CPU01_CONN2_DATA.SEND_REQ := FALSE;
       #CONN4_SendReq_Dn := FALSE;
       #CPU01_CONN2_DATA.CONN_SETA := FALSE;
       #CPU01_CONN2_DATA.DISCONNECT := FALSE;
       #CPU01_CONN2_DATA.ABORT_REQ := FALSE;
   END_IF;
END_REGION

REGION Network 94: CPU01 Conn2-Establish or register ISO-on_TCP connection
   // After the connection has been established, it is automatically monitored and 
   // maintained by the operating system of the CPU.
   // 
   // If the connection has been interrupted, by any line break or due to the remote 
   // communications partner, the active partner attempts to reestablish the 
   // connection.
   // 
   // Therefore, the FB 65 "TCON" may not be called again!
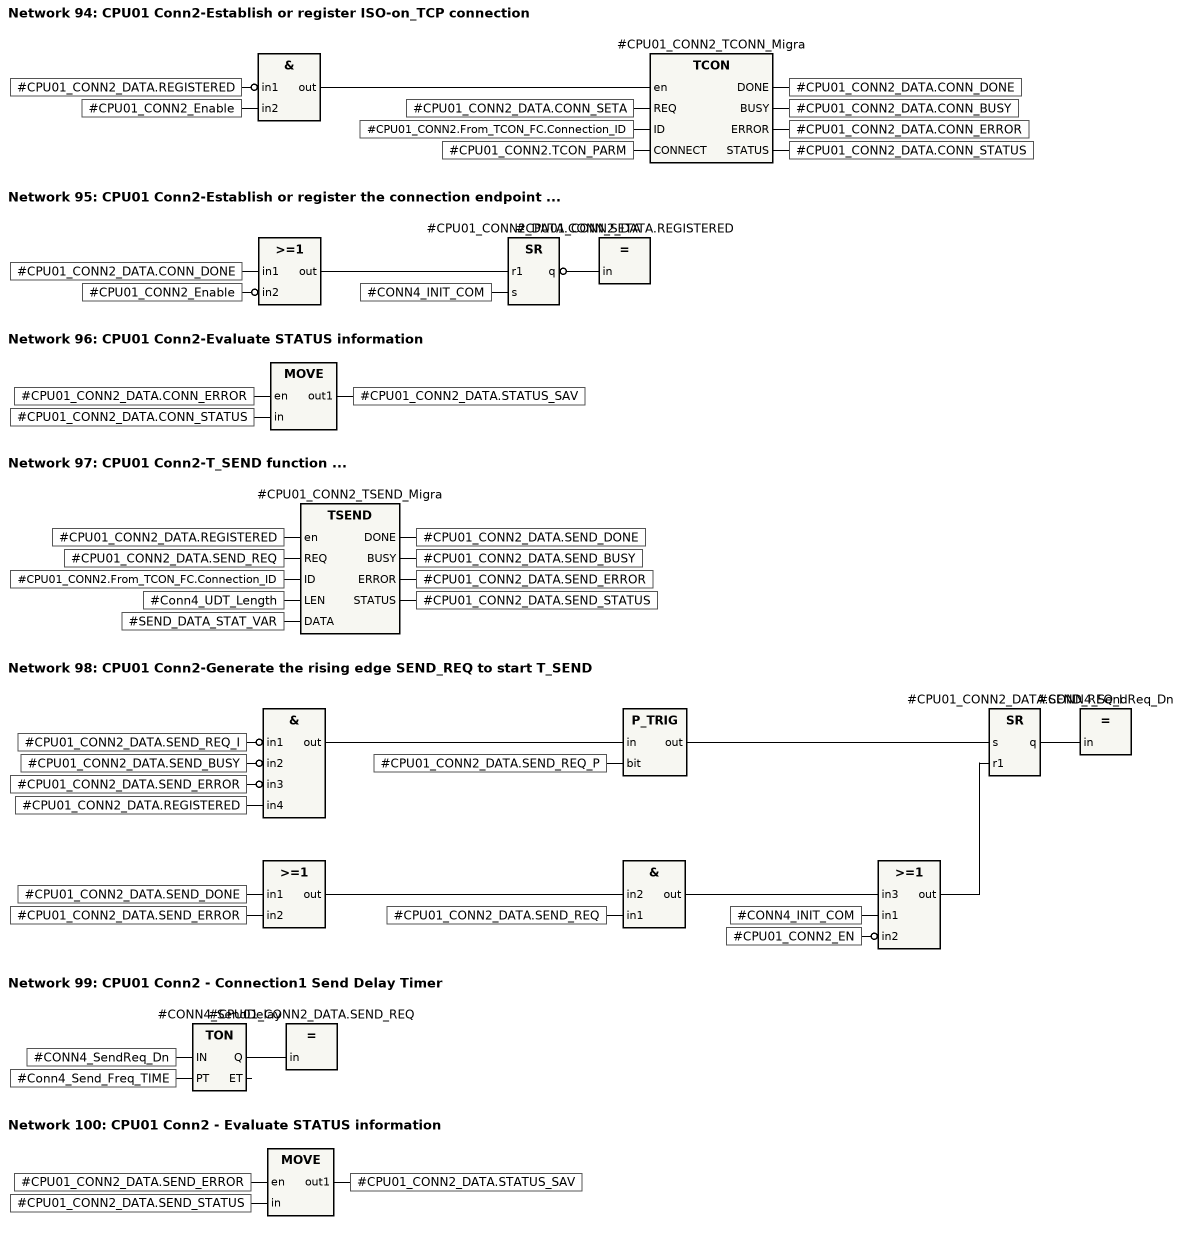
   IF NOT #CPU01_CONN2_DATA.REGISTERED AND #CPU01_CONN2_Enable THEN
       #CPU01_CONN2_TCONN_Migra(REQ := #CPU01_CONN2_DATA.CONN_SETA,   // TCON
                               ID := #CPU01_CONN2.From_TCON_FC.Connection_ID,
                               CONNECT := #CPU01_CONN2.TCON_PARM,
                               DONE => #CPU01_CONN2_DATA.CONN_DONE,
                               BUSY => #CPU01_CONN2_DATA.CONN_BUSY,
                               ERROR => #CPU01_CONN2_DATA.CONN_ERROR,
                               STATUS => #CPU01_CONN2_DATA.CONN_STATUS);
   END_IF;
END_REGION

REGION Network 95: CPU01 Conn2-Establish or register the connection endpoint ...
   // while startup phase (initial).
   // 
   // Indication of the connection status:
   // 
   // a) If the CPU may establish the specified connection after Stop/Run  
   // immediately, the variable "REGISTERED" indicates HIGH (=1).
   // 
   // b) If the CPU is not able to establish the specified connection after Stop/Run, 
   // the variable "REGISTERED" remains LOW(=0).
   // 
   // c) Note: If the instance DB is loaded by the user, the variable "REGISTERED" 
   // indicates HIGH, although the connection may not be established yet. 
   // However, the FB64 "TRCV" would indicate the STATUS=0x80C4, as long as the 
   // connection has not been established.
   IF #CONN4_INIT_COM THEN
       #CPU01_CONN2_DATA.CONN_SETA := TRUE;   // SR flip-flop
   END_IF;
   IF #CPU01_CONN2_DATA.CONN_DONE OR NOT #CPU01_CONN2_Enable THEN
       #CPU01_CONN2_DATA.CONN_SETA := FALSE;
   END_IF;
   #CPU01_CONN2_DATA.REGISTERED := NOT #CPU01_CONN2_DATA.CONN_SETA;
END_REGION

REGION Network 96: CPU01 Conn2-Evaluate STATUS information
   // If ERROR occured then save STATUS!
   IF #CPU01_CONN2_DATA.CONN_ERROR THEN
       #CPU01_CONN2_DATA.STATUS_SAV := #CPU01_CONN2_DATA.CONN_STATUS;
   END_IF;
END_REGION

REGION Network 97: CPU01 Conn2-T_SEND function ...
   // if connection is established to transmit the data to the partner as a message.
   IF #CPU01_CONN2_DATA.REGISTERED THEN
       #CPU01_CONN2_TSEND_Migra(REQ := #CPU01_CONN2_DATA.SEND_REQ,   // TSEND
                               ID := #CPU01_CONN2.From_TCON_FC.Connection_ID,
                               LEN := #Conn4_UDT_Length,
                               DATA := #SEND_DATA_STAT_VAR,
                               DONE => #CPU01_CONN2_DATA.SEND_DONE,
                               BUSY => #CPU01_CONN2_DATA.SEND_BUSY,
                               ERROR => #CPU01_CONN2_DATA.SEND_ERROR,
                               STATUS => #CPU01_CONN2_DATA.SEND_STATUS);
   END_IF;
END_REGION

REGION Network 98: CPU01 Conn2-Generate the rising edge SEND_REQ to start T_SEND
   #_w1 := NOT #CPU01_CONN2_DATA.SEND_REQ_I AND NOT #CPU01_CONN2_DATA.SEND_BUSY AND NOT #CPU01_CONN2_DATA.SEND_ERROR AND #CPU01_CONN2_DATA.REGISTERED;
   #_w2 := #_w1 AND NOT #CPU01_CONN2_DATA.SEND_REQ_P;   // rising edge
   #CPU01_CONN2_DATA.SEND_REQ_P := #_w1;
   IF #_w2 THEN
       #CPU01_CONN2_DATA.SEND_REQ_I := TRUE;   // SR flip-flop
   END_IF;
   IF ((#CPU01_CONN2_DATA.SEND_DONE OR #CPU01_CONN2_DATA.SEND_ERROR) AND #CPU01_CONN2_DATA.SEND_REQ) OR #CONN4_INIT_COM OR NOT #CPU01_CONN2_EN THEN
       #CPU01_CONN2_DATA.SEND_REQ_I := FALSE;
   END_IF;
   #CONN4_SendReq_Dn := #CPU01_CONN2_DATA.SEND_REQ_I;
END_REGION

REGION Network 99: CPU01 Conn2 - Connection1 Send Delay Timer
   #CONN4_SendDelay(IN := #CONN4_SendReq_Dn, PT := #Conn4_Send_Freq_TIME);   // TON
   #CPU01_CONN2_DATA.SEND_REQ := #CONN4_SendDelay.Q;
END_REGION

REGION Network 100: CPU01 Conn2 - Evaluate STATUS information
   // If ERROR occured then save STATUS!
   IF #CPU01_CONN2_DATA.SEND_ERROR THEN
       #CPU01_CONN2_DATA.STATUS_SAV := #CPU01_CONN2_DATA.SEND_STATUS;
   END_IF;
END_REGION

REGION Network 101: CPU01 Conn2 -TCON Receive Block
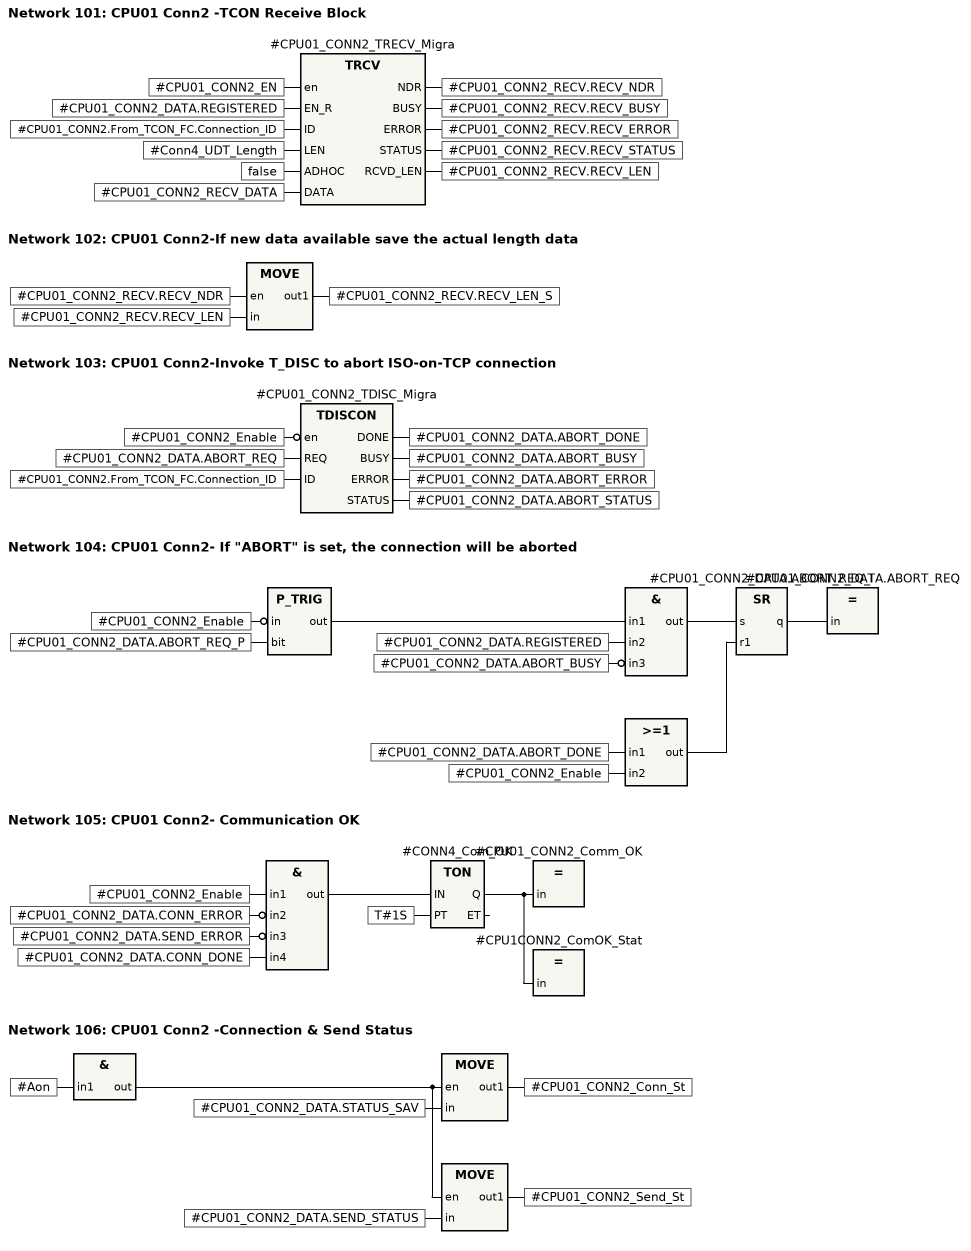
   IF #CPU01_CONN2_EN THEN
       #CPU01_CONN2_TRECV_Migra(EN_R := #CPU01_CONN2_DATA.REGISTERED,   // TRCV
                               ID := #CPU01_CONN2.From_TCON_FC.Connection_ID,
                               LEN := #Conn4_UDT_Length,
                               ADHOC := false,
                               DATA := #CPU01_CONN2_RECV_DATA,
                               NDR => #CPU01_CONN2_RECV.RECV_NDR,
                               BUSY => #CPU01_CONN2_RECV.RECV_BUSY,
                               ERROR => #CPU01_CONN2_RECV.RECV_ERROR,
                               STATUS => #CPU01_CONN2_RECV.RECV_STATUS,
                               RCVD_LEN => #CPU01_CONN2_RECV.RECV_LEN);
   END_IF;
END_REGION

REGION Network 102: CPU01 Conn2-If new data available save the actual length data
   IF #CPU01_CONN2_RECV.RECV_NDR THEN #CPU01_CONN2_RECV.RECV_LEN_S := #CPU01_CONN2_RECV.RECV_LEN; END_IF;
END_REGION

REGION Network 103: CPU01 Conn2-Invoke T_DISC to abort ISO-on-TCP connection
   // The FB 66 "TDISCON" terminates a communications connection from the CPU to a
   // communications partner.
   // 
   // An existing connection is terminated when FB 66 "TDISCON" is called or when the
   // CPU has gone into STOP mode. To reestablish the connection, the FB 65 "TCON" 
   // has to be invoked again.
   IF NOT #CPU01_CONN2_Enable THEN
       #CPU01_CONN2_TDISC_Migra(REQ := #CPU01_CONN2_DATA.ABORT_REQ,   // TDISCON
                               ID := #CPU01_CONN2.From_TCON_FC.Connection_ID,
                               DONE => #CPU01_CONN2_DATA.ABORT_DONE,
                               BUSY => #CPU01_CONN2_DATA.ABORT_BUSY,
                               ERROR => #CPU01_CONN2_DATA.ABORT_ERROR,
                               STATUS => #CPU01_CONN2_DATA.ABORT_STATUS);
   END_IF;
END_REGION

REGION Network 104: CPU01 Conn2- If "ABORT" is set, the connection will be aborted
   #_w1 := NOT #CPU01_CONN2_Enable AND NOT #CPU01_CONN2_DATA.ABORT_REQ_P;   // rising edge
   #CPU01_CONN2_DATA.ABORT_REQ_P := NOT #CPU01_CONN2_Enable;
   IF #_w1 AND #CPU01_CONN2_DATA.REGISTERED AND NOT #CPU01_CONN2_DATA.ABORT_BUSY THEN
       #CPU01_CONN2_DATA.ABORT_REQ_I := TRUE;   // SR flip-flop
   END_IF;
   IF #CPU01_CONN2_DATA.ABORT_DONE OR #CPU01_CONN2_Enable THEN
       #CPU01_CONN2_DATA.ABORT_REQ_I := FALSE;
   END_IF;
   #CPU01_CONN2_DATA.ABORT_REQ := #CPU01_CONN2_DATA.ABORT_REQ_I;
END_REGION

REGION Network 105: CPU01 Conn2- Communication OK
   #CONN4_Com_OK(IN := #CPU01_CONN2_Enable AND NOT #CPU01_CONN2_DATA.CONN_ERROR AND NOT #CPU01_CONN2_DATA.SEND_ERROR AND #CPU01_CONN2_DATA.CONN_DONE,   // TON
                 PT := T#1S);
   #CPU01_CONN2_Comm_OK := #CONN4_Com_OK.Q;
   #CPU1CONN2_ComOK_Stat := #CONN4_Com_OK.Q;
END_REGION

REGION Network 106: CPU01 Conn2 -Connection & Send Status
   IF #Aon THEN
       #CPU01_CONN2_Conn_St := #CPU01_CONN2_DATA.STATUS_SAV;
       #CPU01_CONN2_Send_St := #CPU01_CONN2_DATA.SEND_STATUS;
   END_IF;
END_REGION

REGION Network 107: CPU01 Connection 2 Receive Status
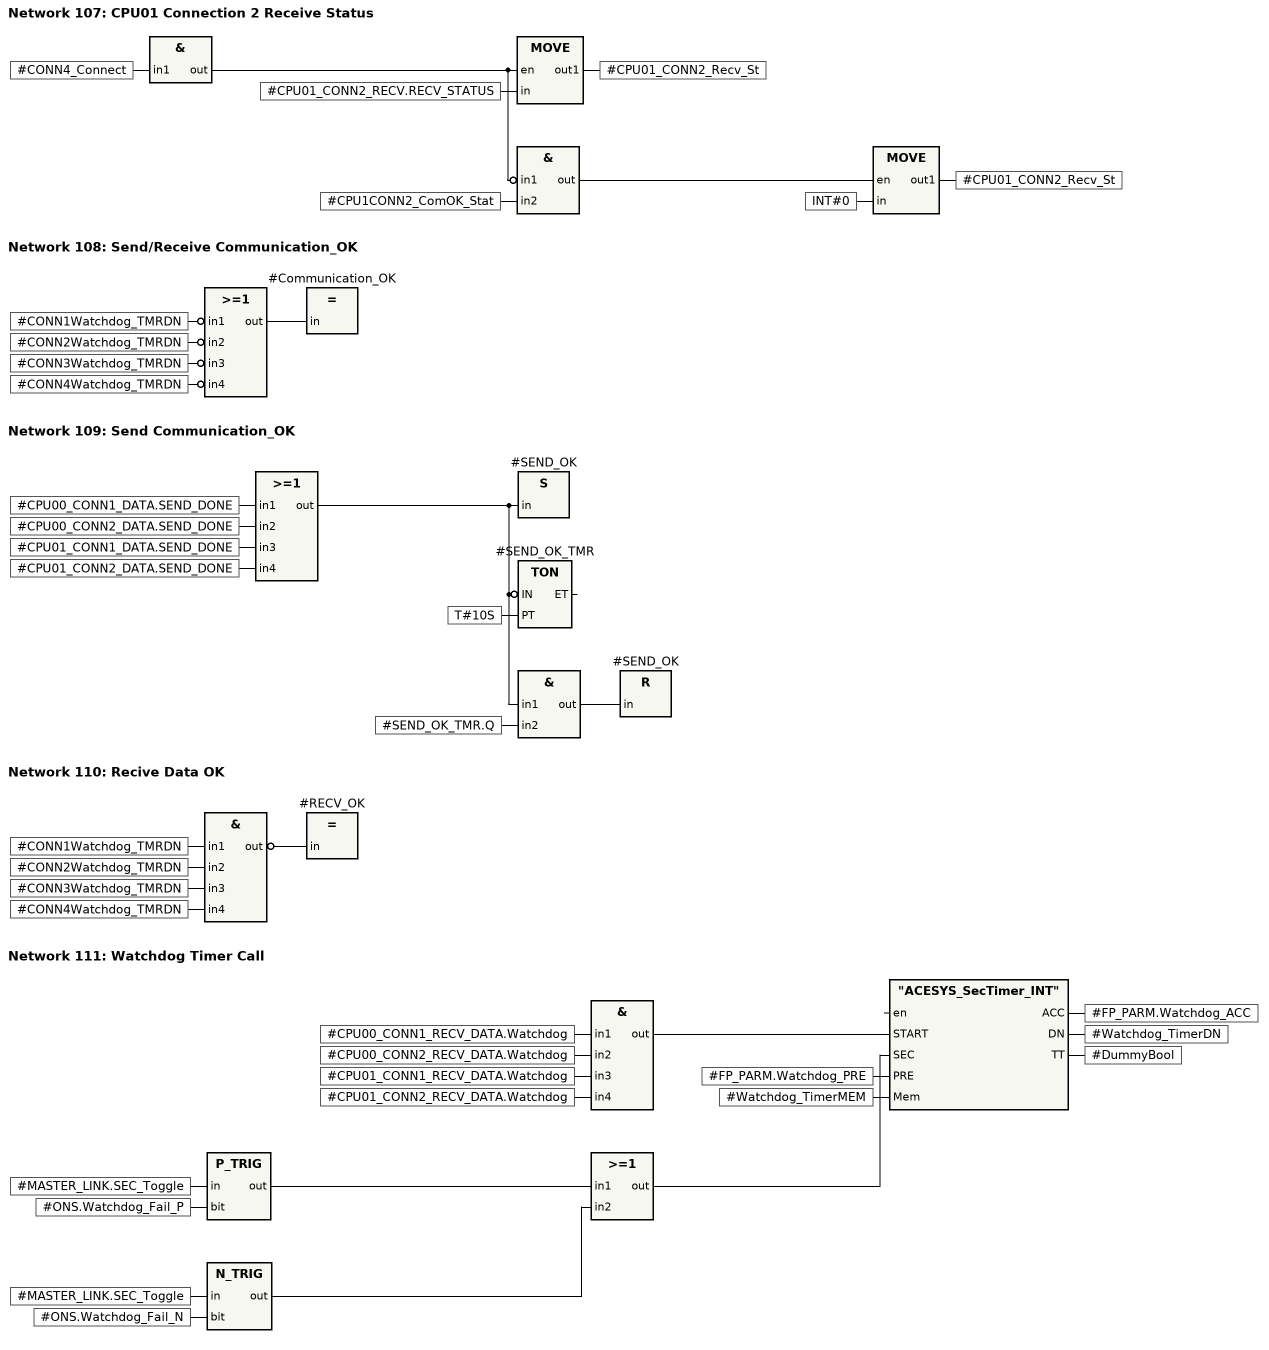
   IF #CONN4_Connect THEN #CPU01_CONN2_Recv_St := #CPU01_CONN2_RECV.RECV_STATUS; END_IF;
   IF NOT #CONN4_Connect AND #CPU1CONN2_ComOK_Stat THEN #CPU01_CONN2_Recv_St := INT#0; END_IF;
END_REGION

REGION Network 108: Send/Receive Communication_OK
   #Communication_OK := NOT #CONN1Watchdog_TMRDN OR NOT #CONN2Watchdog_TMRDN OR NOT #CONN3Watchdog_TMRDN OR NOT #CONN4Watchdog_TMRDN;
END_REGION

REGION Network 109: Send Communication_OK
   #_w1 := #CPU00_CONN1_DATA.SEND_DONE OR #CPU00_CONN2_DATA.SEND_DONE OR #CPU01_CONN1_DATA.SEND_DONE OR #CPU01_CONN2_DATA.SEND_DONE;
   IF #_w1 THEN #SEND_OK := TRUE; END_IF;
   #SEND_OK_TMR(IN := NOT #_w1, PT := T#10S);   // TON
   IF #_w1 AND #SEND_OK_TMR.Q THEN #SEND_OK := FALSE; END_IF;
END_REGION

REGION Network 110: Recive Data OK
   #RECV_OK := NOT (#CONN1Watchdog_TMRDN AND #CONN2Watchdog_TMRDN AND #CONN3Watchdog_TMRDN AND #CONN4Watchdog_TMRDN);
END_REGION

REGION Network 111: Watchdog Timer Call
   #_w1 := #MASTER_LINK.SEC_Toggle AND NOT #ONS.Watchdog_Fail_P;   // rising edge
   #ONS.Watchdog_Fail_P := #MASTER_LINK.SEC_Toggle;
   #_w2 := NOT #MASTER_LINK.SEC_Toggle AND #ONS.Watchdog_Fail_N;   // falling edge
   #ONS.Watchdog_Fail_N := #MASTER_LINK.SEC_Toggle;
   "ACESYS_SecTimer_INT"(START := #CPU00_CONN1_RECV_DATA.Watchdog AND #CPU00_CONN2_RECV_DATA.Watchdog AND #CPU01_CONN1_RECV_DATA.Watchdog AND #CPU01_CONN2_RECV_DATA.Watchdog,
                         SEC := #_w1 OR #_w2,
                         PRE := #FP_PARM.Watchdog_PRE,
                         Mem := #Watchdog_TimerMEM,
                         ACC => #FP_PARM.Watchdog_ACC,
                         DN => #Watchdog_TimerDN,
                         TT => #DummyBool);
END_REGION

REGION Network 112: CPU00 Connection 1 Watchdog Timer Call
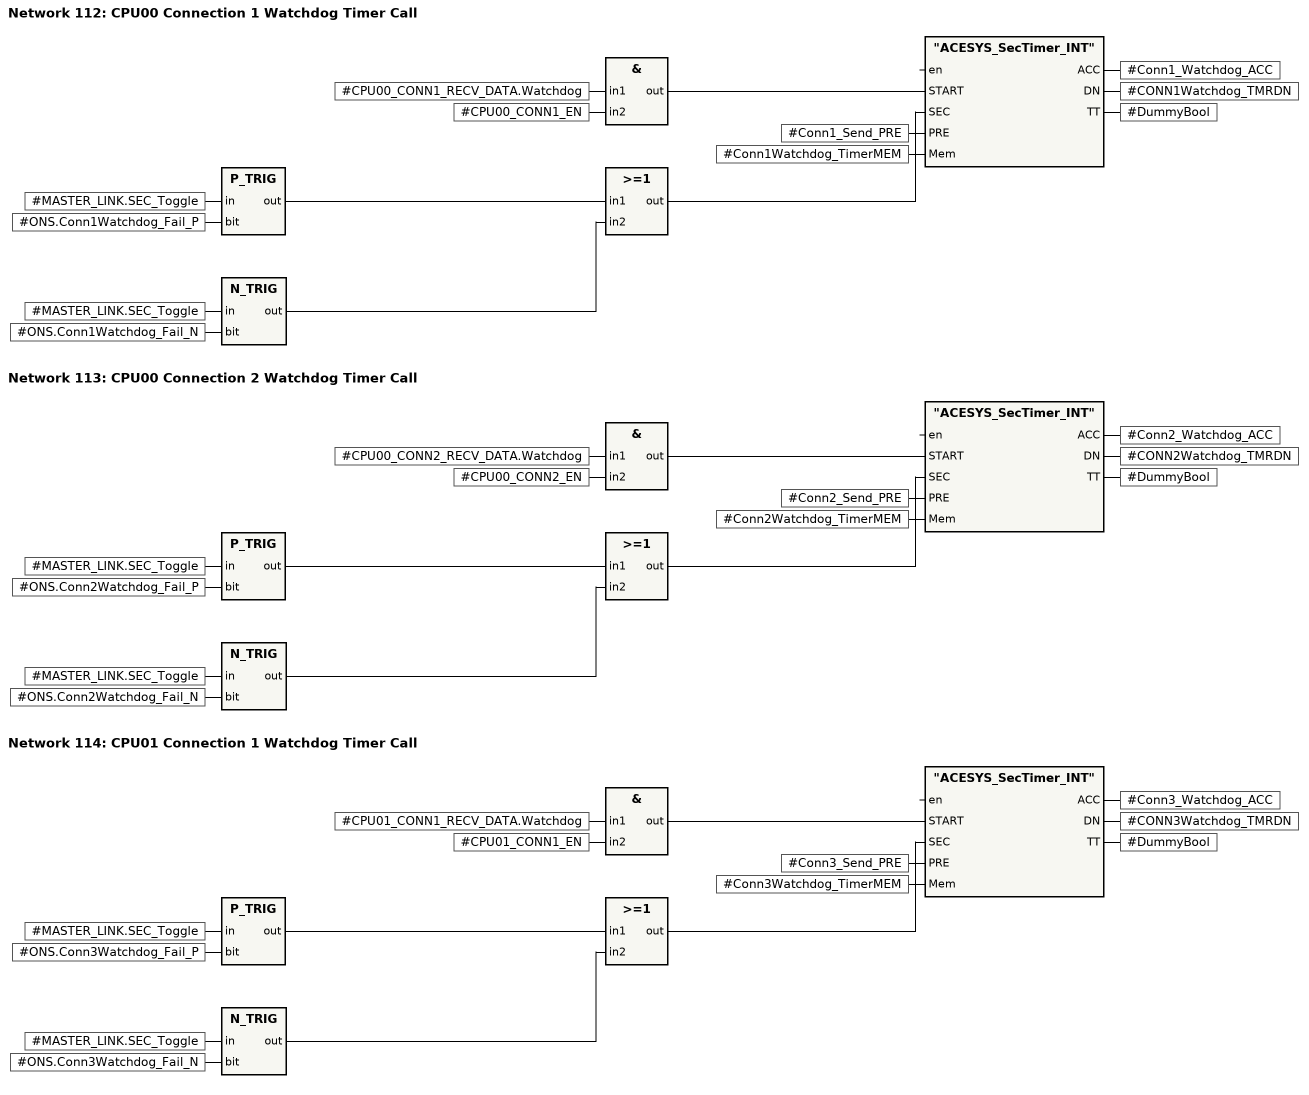
   #_w1 := #MASTER_LINK.SEC_Toggle AND NOT #ONS.Conn1Watchdog_Fail_P;   // rising edge
   #ONS.Conn1Watchdog_Fail_P := #MASTER_LINK.SEC_Toggle;
   #_w2 := NOT #MASTER_LINK.SEC_Toggle AND #ONS.Conn1Watchdog_Fail_N;   // falling edge
   #ONS.Conn1Watchdog_Fail_N := #MASTER_LINK.SEC_Toggle;
   "ACESYS_SecTimer_INT"(START := #CPU00_CONN1_RECV_DATA.Watchdog AND #CPU00_CONN1_EN,
                         SEC := #_w1 OR #_w2,
                         PRE := #Conn1_Send_PRE,
                         Mem := #Conn1Watchdog_TimerMEM,
                         ACC => #Conn1_Watchdog_ACC,
                         DN => #CONN1Watchdog_TMRDN,
                         TT => #DummyBool);
END_REGION

REGION Network 113: CPU00 Connection 2 Watchdog Timer Call
   #_w1 := #MASTER_LINK.SEC_Toggle AND NOT #ONS.Conn2Watchdog_Fail_P;   // rising edge
   #ONS.Conn2Watchdog_Fail_P := #MASTER_LINK.SEC_Toggle;
   #_w2 := NOT #MASTER_LINK.SEC_Toggle AND #ONS.Conn2Watchdog_Fail_N;   // falling edge
   #ONS.Conn2Watchdog_Fail_N := #MASTER_LINK.SEC_Toggle;
   "ACESYS_SecTimer_INT"(START := #CPU00_CONN2_RECV_DATA.Watchdog AND #CPU00_CONN2_EN,
                         SEC := #_w1 OR #_w2,
                         PRE := #Conn2_Send_PRE,
                         Mem := #Conn2Watchdog_TimerMEM,
                         ACC => #Conn2_Watchdog_ACC,
                         DN => #CONN2Watchdog_TMRDN,
                         TT => #DummyBool);
END_REGION

REGION Network 114: CPU01 Connection 1 Watchdog Timer Call
   #_w1 := #MASTER_LINK.SEC_Toggle AND NOT #ONS.Conn3Watchdog_Fail_P;   // rising edge
   #ONS.Conn3Watchdog_Fail_P := #MASTER_LINK.SEC_Toggle;
   #_w2 := NOT #MASTER_LINK.SEC_Toggle AND #ONS.Conn3Watchdog_Fail_N;   // falling edge
   #ONS.Conn3Watchdog_Fail_N := #MASTER_LINK.SEC_Toggle;
   "ACESYS_SecTimer_INT"(START := #CPU01_CONN1_RECV_DATA.Watchdog AND #CPU01_CONN1_EN,
                         SEC := #_w1 OR #_w2,
                         PRE := #Conn3_Send_PRE,
                         Mem := #Conn3Watchdog_TimerMEM,
                         ACC => #Conn3_Watchdog_ACC,
                         DN => #CONN3Watchdog_TMRDN,
                         TT => #DummyBool);
END_REGION

REGION Network 115: CPU01 Connection 2 Watchdog Timer Call
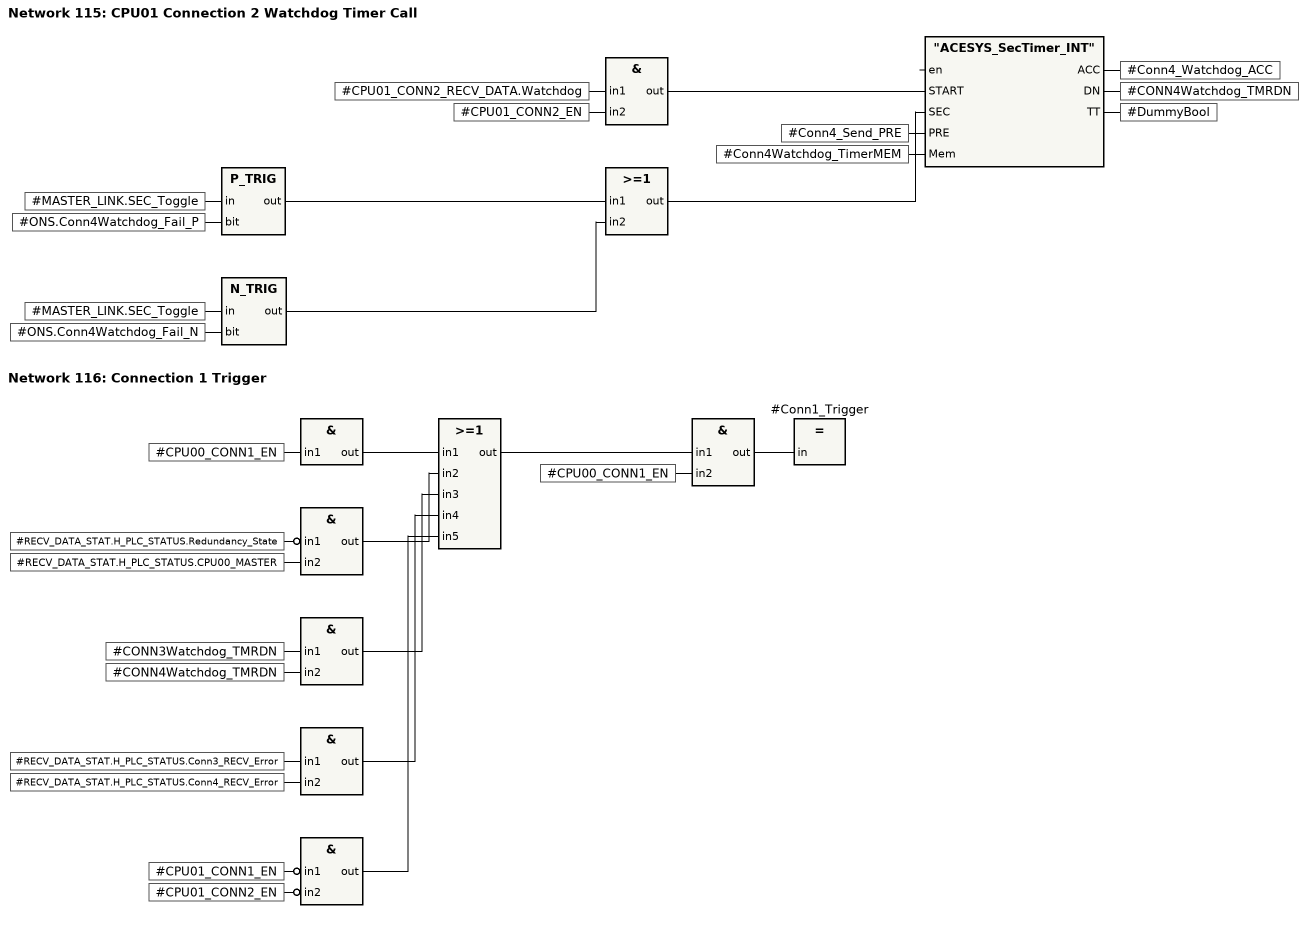
   #_w1 := #MASTER_LINK.SEC_Toggle AND NOT #ONS.Conn4Watchdog_Fail_P;   // rising edge
   #ONS.Conn4Watchdog_Fail_P := #MASTER_LINK.SEC_Toggle;
   #_w2 := NOT #MASTER_LINK.SEC_Toggle AND #ONS.Conn4Watchdog_Fail_N;   // falling edge
   #ONS.Conn4Watchdog_Fail_N := #MASTER_LINK.SEC_Toggle;
   "ACESYS_SecTimer_INT"(START := #CPU01_CONN2_RECV_DATA.Watchdog AND #CPU01_CONN2_EN,
                         SEC := #_w1 OR #_w2,
                         PRE := #Conn4_Send_PRE,
                         Mem := #Conn4Watchdog_TimerMEM,
                         ACC => #Conn4_Watchdog_ACC,
                         DN => #CONN4Watchdog_TMRDN,
                         TT => #DummyBool);
END_REGION

REGION Network 116: Connection 1 Trigger
   #Conn1_Trigger := (#CPU00_CONN1_EN OR (NOT #RECV_DATA_STAT.H_PLC_STATUS.Redundancy_State AND #RECV_DATA_STAT.H_PLC_STATUS.CPU00_MASTER) OR (#CONN3Watchdog_TMRDN AND #CONN4Watchdog_TMRDN) OR (#RECV_DATA_STAT.H_PLC_STATUS.Conn3_RECV_Error AND #RECV_DATA_STAT.H_PLC_STATUS.Conn4_RECV_Error) OR (NOT #CPU01_CONN1_EN AND NOT #CPU01_CONN2_EN)) AND #CPU00_CONN1_EN;
END_REGION

REGION Network 117: Connection 2 Trigger
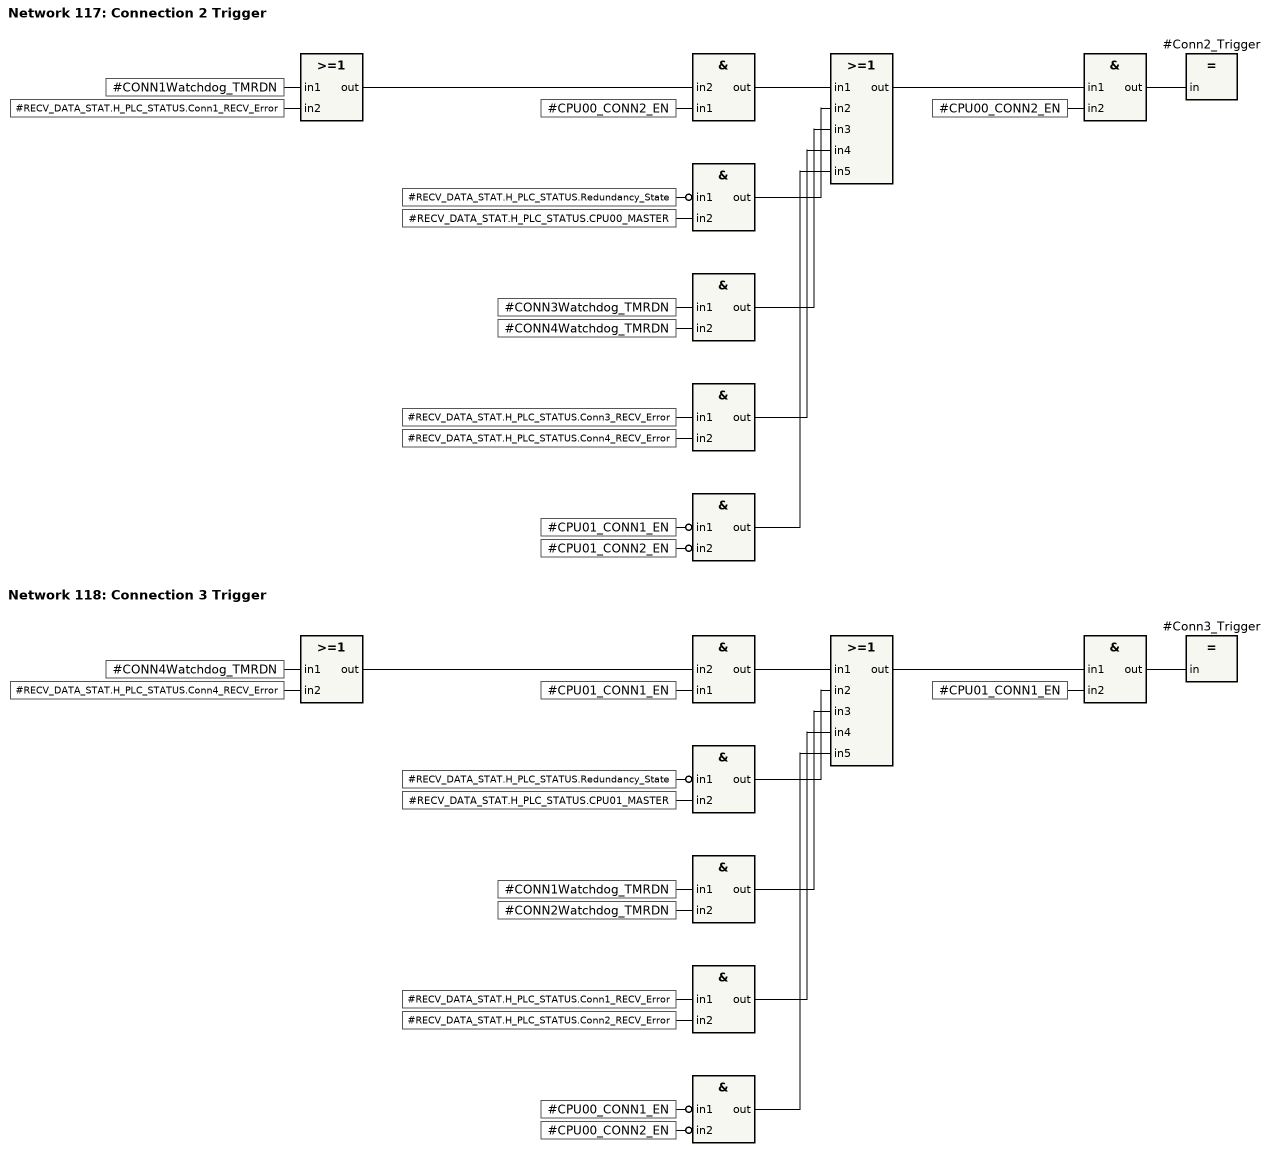
   #Conn2_Trigger := (((#CONN1Watchdog_TMRDN OR #RECV_DATA_STAT.H_PLC_STATUS.Conn1_RECV_Error) AND #CPU00_CONN2_EN) OR (NOT #RECV_DATA_STAT.H_PLC_STATUS.Redundancy_State AND #RECV_DATA_STAT.H_PLC_STATUS.CPU00_MASTER) OR (#CONN3Watchdog_TMRDN AND #CONN4Watchdog_TMRDN) OR (#RECV_DATA_STAT.H_PLC_STATUS.Conn3_RECV_Error AND #RECV_DATA_STAT.H_PLC_STATUS.Conn4_RECV_Error) OR (NOT #CPU01_CONN1_EN AND NOT #CPU01_CONN2_EN)) AND #CPU00_CONN2_EN;
END_REGION

REGION Network 118: Connection 3 Trigger
   #Conn3_Trigger := (((#CONN4Watchdog_TMRDN OR #RECV_DATA_STAT.H_PLC_STATUS.Conn4_RECV_Error) AND #CPU01_CONN1_EN) OR (NOT #RECV_DATA_STAT.H_PLC_STATUS.Redundancy_State AND #RECV_DATA_STAT.H_PLC_STATUS.CPU01_MASTER) OR (#CONN1Watchdog_TMRDN AND #CONN2Watchdog_TMRDN) OR (#RECV_DATA_STAT.H_PLC_STATUS.Conn1_RECV_Error AND #RECV_DATA_STAT.H_PLC_STATUS.Conn2_RECV_Error) OR (NOT #CPU00_CONN1_EN AND NOT #CPU00_CONN2_EN)) AND #CPU01_CONN1_EN;
END_REGION

REGION Network 119: Connection 4 Trigger
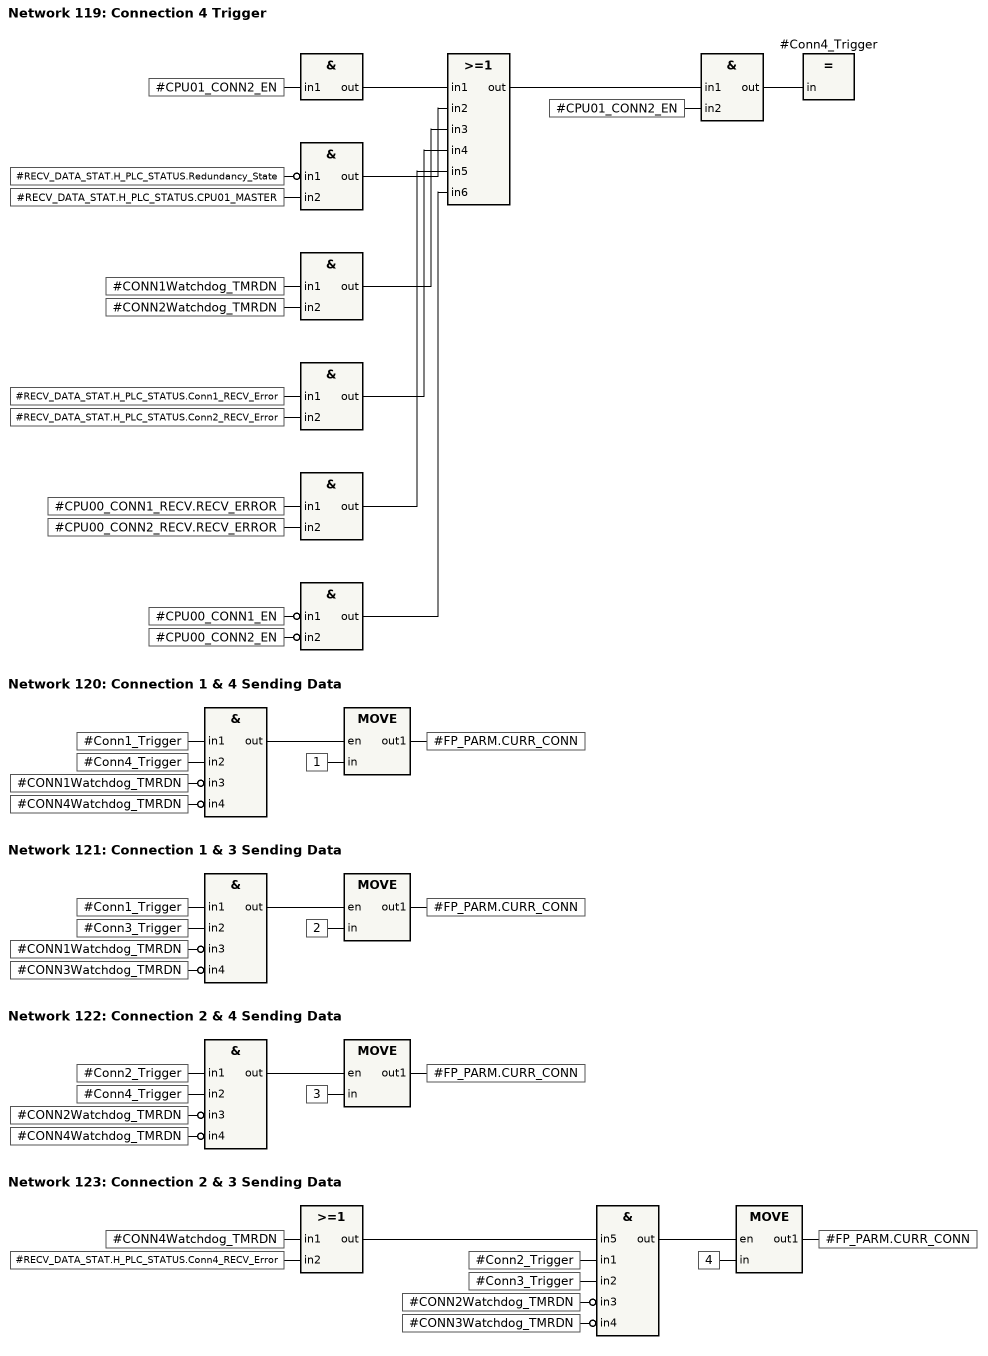
   #Conn4_Trigger := (#CPU01_CONN2_EN OR (NOT #RECV_DATA_STAT.H_PLC_STATUS.Redundancy_State AND #RECV_DATA_STAT.H_PLC_STATUS.CPU01_MASTER) OR (#CONN1Watchdog_TMRDN AND #CONN2Watchdog_TMRDN) OR (#RECV_DATA_STAT.H_PLC_STATUS.Conn1_RECV_Error AND #RECV_DATA_STAT.H_PLC_STATUS.Conn2_RECV_Error) OR (#CPU00_CONN1_RECV.RECV_ERROR AND #CPU00_CONN2_RECV.RECV_ERROR) OR (NOT #CPU00_CONN1_EN AND NOT #CPU00_CONN2_EN)) AND #CPU01_CONN2_EN;
END_REGION

REGION Network 120: Connection 1 & 4 Sending Data
   IF #Conn1_Trigger AND #Conn4_Trigger AND NOT #CONN1Watchdog_TMRDN AND NOT #CONN4Watchdog_TMRDN THEN
       #FP_PARM.CURR_CONN := 1;
   END_IF;
END_REGION

REGION Network 121: Connection 1 & 3 Sending Data
   IF #Conn1_Trigger AND #Conn3_Trigger AND NOT #CONN1Watchdog_TMRDN AND NOT #CONN3Watchdog_TMRDN THEN
       #FP_PARM.CURR_CONN := 2;
   END_IF;
END_REGION

REGION Network 122: Connection 2 & 4 Sending Data
   IF #Conn2_Trigger AND #Conn4_Trigger AND NOT #CONN2Watchdog_TMRDN AND NOT #CONN4Watchdog_TMRDN THEN
       #FP_PARM.CURR_CONN := 3;
   END_IF;
END_REGION

REGION Network 123: Connection 2 & 3 Sending Data
   IF (#CONN4Watchdog_TMRDN OR #RECV_DATA_STAT.H_PLC_STATUS.Conn4_RECV_Error) AND #Conn2_Trigger AND #Conn3_Trigger AND NOT #CONN2Watchdog_TMRDN AND NOT #CONN3Watchdog_TMRDN THEN
       #FP_PARM.CURR_CONN := 4;
   END_IF;
END_REGION

REGION Network 124: Individual Connection 1
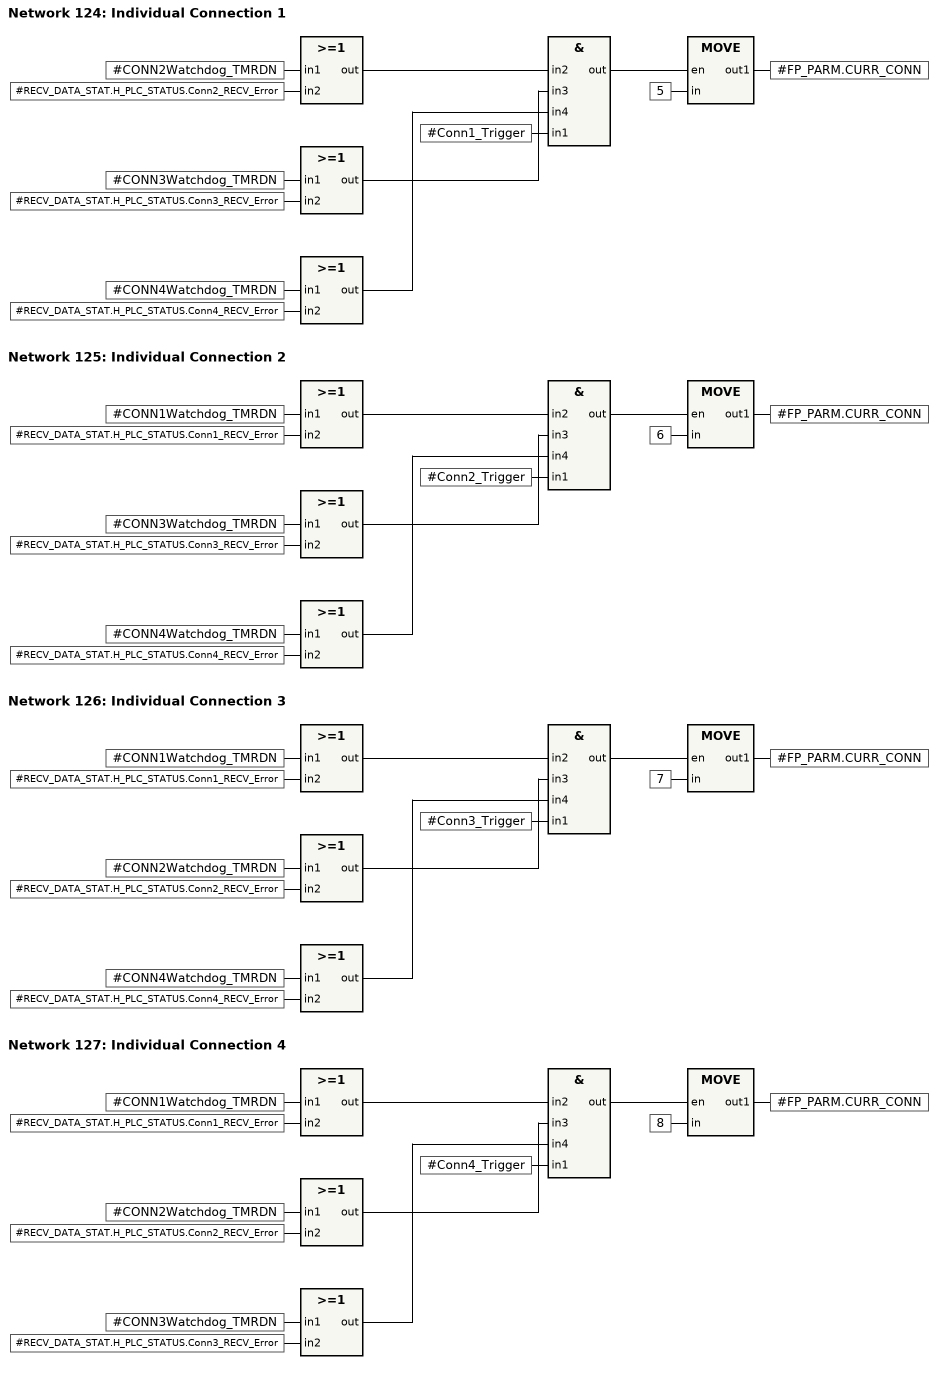
   IF (#CONN2Watchdog_TMRDN OR #RECV_DATA_STAT.H_PLC_STATUS.Conn2_RECV_Error) AND (#CONN3Watchdog_TMRDN OR #RECV_DATA_STAT.H_PLC_STATUS.Conn3_RECV_Error) AND (#CONN4Watchdog_TMRDN OR #RECV_DATA_STAT.H_PLC_STATUS.Conn4_RECV_Error) AND #Conn1_Trigger THEN
       #FP_PARM.CURR_CONN := 5;
   END_IF;
END_REGION

REGION Network 125: Individual Connection 2
   IF (#CONN1Watchdog_TMRDN OR #RECV_DATA_STAT.H_PLC_STATUS.Conn1_RECV_Error) AND (#CONN3Watchdog_TMRDN OR #RECV_DATA_STAT.H_PLC_STATUS.Conn3_RECV_Error) AND (#CONN4Watchdog_TMRDN OR #RECV_DATA_STAT.H_PLC_STATUS.Conn4_RECV_Error) AND #Conn2_Trigger THEN
       #FP_PARM.CURR_CONN := 6;
   END_IF;
END_REGION

REGION Network 126: Individual Connection 3
   IF (#CONN1Watchdog_TMRDN OR #RECV_DATA_STAT.H_PLC_STATUS.Conn1_RECV_Error) AND (#CONN2Watchdog_TMRDN OR #RECV_DATA_STAT.H_PLC_STATUS.Conn2_RECV_Error) AND (#CONN4Watchdog_TMRDN OR #RECV_DATA_STAT.H_PLC_STATUS.Conn4_RECV_Error) AND #Conn3_Trigger THEN
       #FP_PARM.CURR_CONN := 7;
   END_IF;
END_REGION

REGION Network 127: Individual Connection 4
   IF (#CONN1Watchdog_TMRDN OR #RECV_DATA_STAT.H_PLC_STATUS.Conn1_RECV_Error) AND (#CONN2Watchdog_TMRDN OR #RECV_DATA_STAT.H_PLC_STATUS.Conn2_RECV_Error) AND (#CONN3Watchdog_TMRDN OR #RECV_DATA_STAT.H_PLC_STATUS.Conn3_RECV_Error) AND #Conn4_Trigger THEN
       #FP_PARM.CURR_CONN := 8;
   END_IF;
END_REGION

REGION Network 128: Conn 3 & 4 Fails or CPU 01 Stop Mode - Connectionn 1 & 2
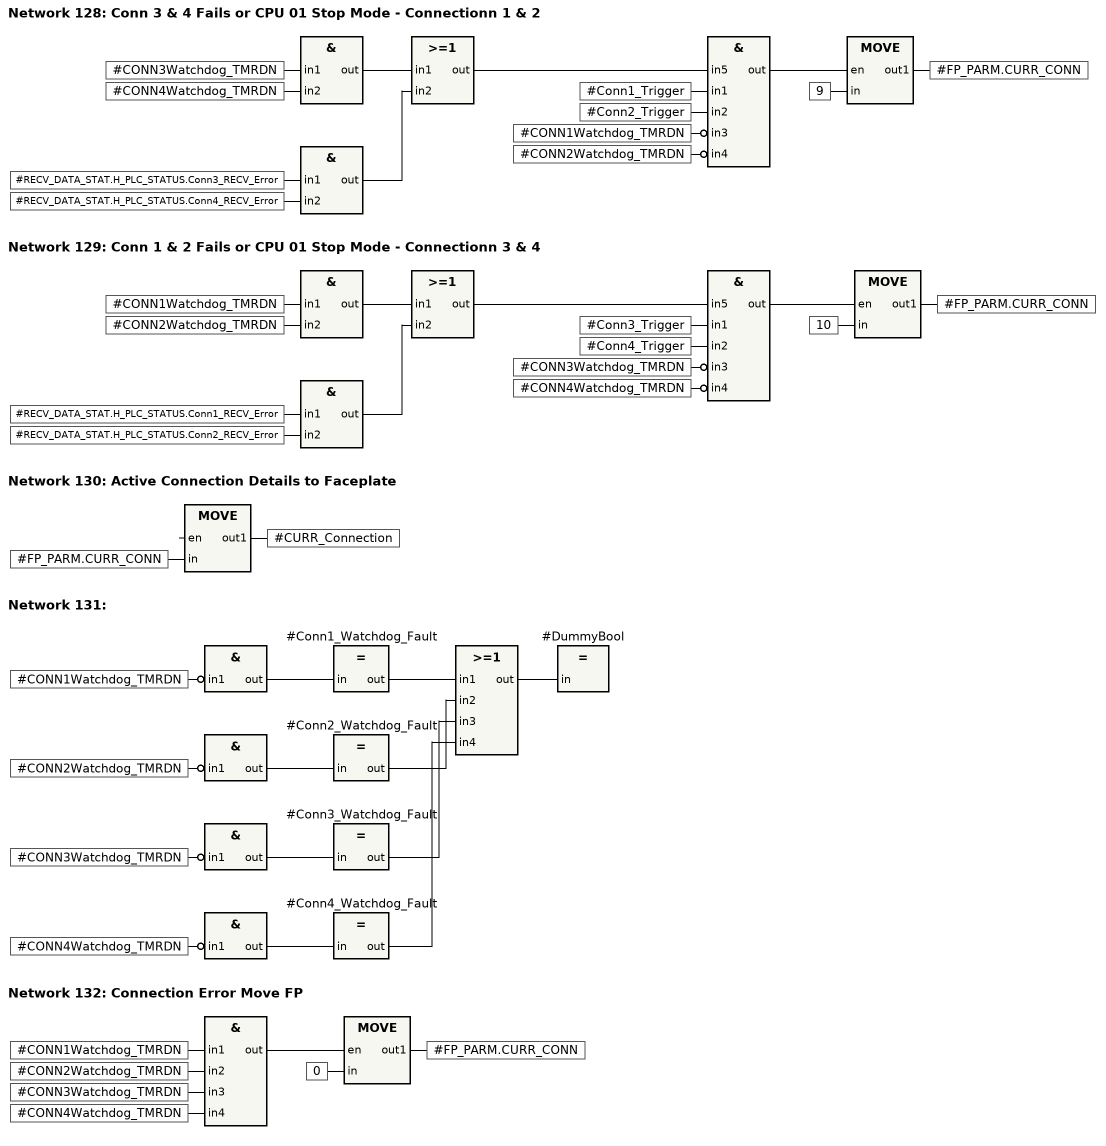
   IF ((#CONN3Watchdog_TMRDN AND #CONN4Watchdog_TMRDN) OR (#RECV_DATA_STAT.H_PLC_STATUS.Conn3_RECV_Error AND #RECV_DATA_STAT.H_PLC_STATUS.Conn4_RECV_Error)) AND #Conn1_Trigger AND #Conn2_Trigger AND NOT #CONN1Watchdog_TMRDN AND NOT #CONN2Watchdog_TMRDN THEN
       #FP_PARM.CURR_CONN := 9;
   END_IF;
END_REGION

REGION Network 129: Conn 1 & 2 Fails or CPU 01 Stop Mode - Connectionn 3 & 4
   IF ((#CONN1Watchdog_TMRDN AND #CONN2Watchdog_TMRDN) OR (#RECV_DATA_STAT.H_PLC_STATUS.Conn1_RECV_Error AND #RECV_DATA_STAT.H_PLC_STATUS.Conn2_RECV_Error)) AND #Conn3_Trigger AND #Conn4_Trigger AND NOT #CONN3Watchdog_TMRDN AND NOT #CONN4Watchdog_TMRDN THEN
       #FP_PARM.CURR_CONN := 10;
   END_IF;
END_REGION

REGION Network 130: Active Connection Details to Faceplate
   #CURR_Connection := #FP_PARM.CURR_CONN;
END_REGION

REGION Network 131
   #Conn1_Watchdog_Fault := NOT #CONN1Watchdog_TMRDN;
   #Conn2_Watchdog_Fault := NOT #CONN2Watchdog_TMRDN;
   #Conn3_Watchdog_Fault := NOT #CONN3Watchdog_TMRDN;
   #Conn4_Watchdog_Fault := NOT #CONN4Watchdog_TMRDN;
   #DummyBool := NOT #CONN1Watchdog_TMRDN OR NOT #CONN2Watchdog_TMRDN OR NOT #CONN3Watchdog_TMRDN OR NOT #CONN4Watchdog_TMRDN;
END_REGION

REGION Network 132: Connection Error Move FP
   IF #CONN1Watchdog_TMRDN AND #CONN2Watchdog_TMRDN AND #CONN3Watchdog_TMRDN AND #CONN4Watchdog_TMRDN THEN
       #FP_PARM.CURR_CONN := 0;
   END_IF;
END_REGION

REGION Network 133: Watchdog Bit Set
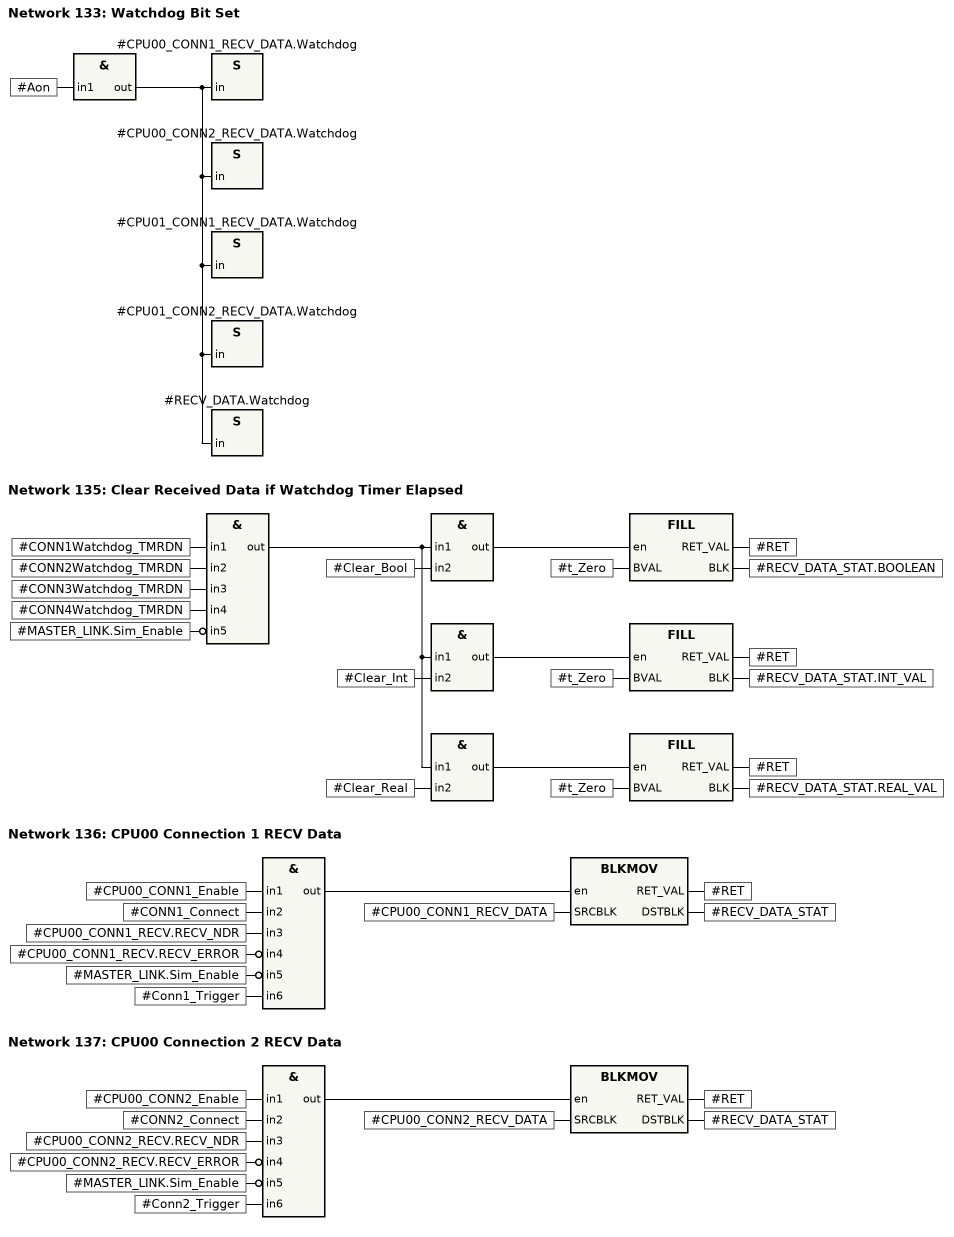
   IF #Aon THEN
       #CPU00_CONN1_RECV_DATA.Watchdog := TRUE;
       #CPU00_CONN2_RECV_DATA.Watchdog := TRUE;
       #CPU01_CONN1_RECV_DATA.Watchdog := TRUE;
       #CPU01_CONN2_RECV_DATA.Watchdog := TRUE;
       #RECV_DATA.Watchdog := TRUE;
   END_IF;
END_REGION

REGION Network 134 (STL): Clear values
         L     0;
         T     #t_Zero;
END_REGION

REGION Network 135: Clear Received Data if Watchdog Timer Elapsed
   #_w1 := #CONN1Watchdog_TMRDN AND #CONN2Watchdog_TMRDN AND #CONN3Watchdog_TMRDN AND #CONN4Watchdog_TMRDN AND NOT #MASTER_LINK.Sim_Enable;
   IF #_w1 AND #Clear_Bool THEN #RET := FILL(BVAL := #t_Zero, BLK => #RECV_DATA_STAT.BOOLEAN); END_IF;
   IF #_w1 AND #Clear_Int THEN #RET := FILL(BVAL := #t_Zero, BLK => #RECV_DATA_STAT.INT_VAL); END_IF;
   IF #_w1 AND #Clear_Real THEN #RET := FILL(BVAL := #t_Zero, BLK => #RECV_DATA_STAT.REAL_VAL); END_IF;
END_REGION

REGION Network 136: CPU00 Connection 1 RECV Data
   IF #CPU00_CONN1_Enable AND #CONN1_Connect AND #CPU00_CONN1_RECV.RECV_NDR AND NOT #CPU00_CONN1_RECV.RECV_ERROR AND NOT #MASTER_LINK.Sim_Enable AND #Conn1_Trigger THEN
       #RET := BLKMOV(SRCBLK := #CPU00_CONN1_RECV_DATA, DSTBLK => #RECV_DATA_STAT);
   END_IF;
END_REGION

REGION Network 137: CPU00 Connection 2 RECV Data
   IF #CPU00_CONN2_Enable AND #CONN2_Connect AND #CPU00_CONN2_RECV.RECV_NDR AND NOT #CPU00_CONN2_RECV.RECV_ERROR AND NOT #MASTER_LINK.Sim_Enable AND #Conn2_Trigger THEN
       #RET := BLKMOV(SRCBLK := #CPU00_CONN2_RECV_DATA, DSTBLK => #RECV_DATA_STAT);
   END_IF;
END_REGION

REGION Network 138: CPU01 Connection 1 RECV Data
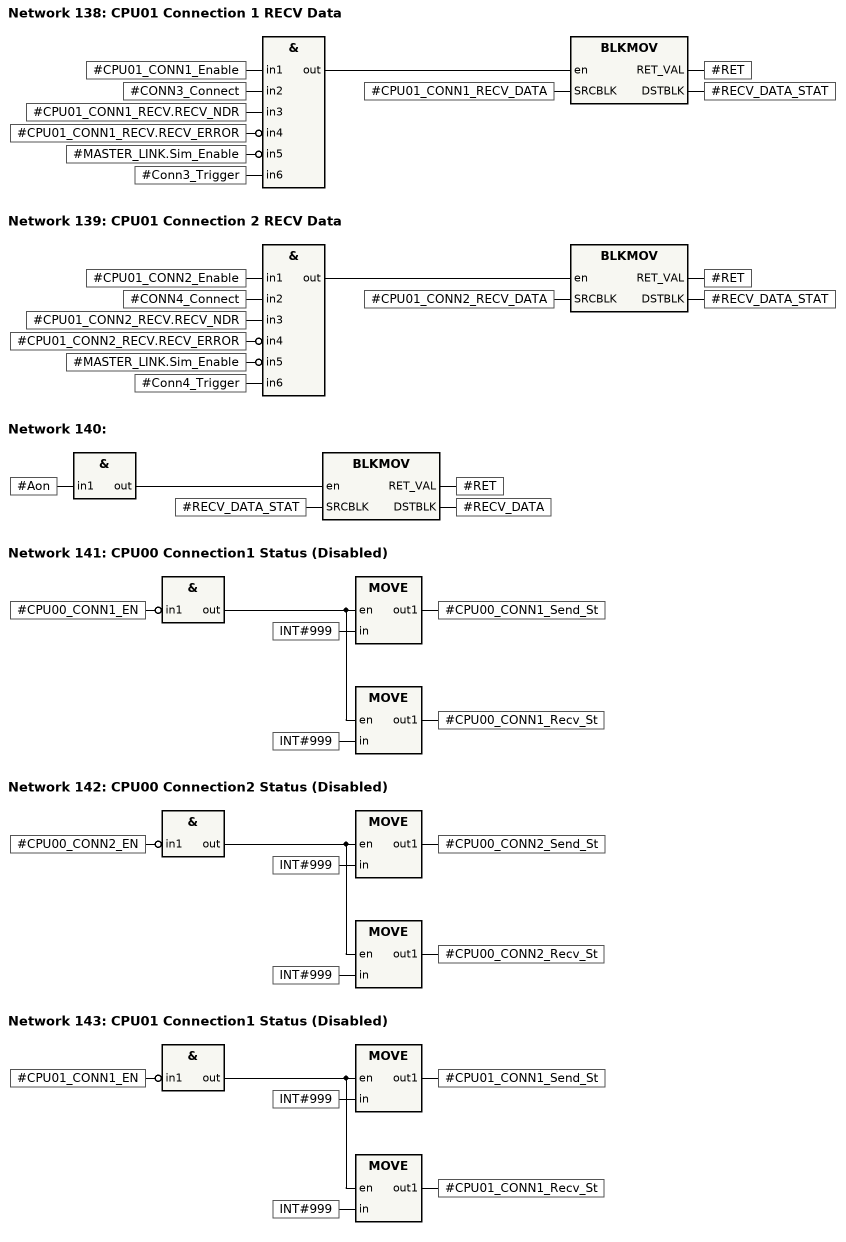
   IF #CPU01_CONN1_Enable AND #CONN3_Connect AND #CPU01_CONN1_RECV.RECV_NDR AND NOT #CPU01_CONN1_RECV.RECV_ERROR AND NOT #MASTER_LINK.Sim_Enable AND #Conn3_Trigger THEN
       #RET := BLKMOV(SRCBLK := #CPU01_CONN1_RECV_DATA, DSTBLK => #RECV_DATA_STAT);
   END_IF;
END_REGION

REGION Network 139: CPU01 Connection 2 RECV Data
   IF #CPU01_CONN2_Enable AND #CONN4_Connect AND #CPU01_CONN2_RECV.RECV_NDR AND NOT #CPU01_CONN2_RECV.RECV_ERROR AND NOT #MASTER_LINK.Sim_Enable AND #Conn4_Trigger THEN
       #RET := BLKMOV(SRCBLK := #CPU01_CONN2_RECV_DATA, DSTBLK => #RECV_DATA_STAT);
   END_IF;
END_REGION

REGION Network 140
   IF #Aon THEN #RET := BLKMOV(SRCBLK := #RECV_DATA_STAT, DSTBLK => #RECV_DATA); END_IF;
END_REGION

REGION Network 141: CPU00 Connection1 Status (Disabled)
   IF NOT #CPU00_CONN1_EN THEN
       #CPU00_CONN1_Send_St := INT#999;
       #CPU00_CONN1_Recv_St := INT#999;
   END_IF;
END_REGION

REGION Network 142: CPU00 Connection2 Status (Disabled)
   IF NOT #CPU00_CONN2_EN THEN
       #CPU00_CONN2_Send_St := INT#999;
       #CPU00_CONN2_Recv_St := INT#999;
   END_IF;
END_REGION

REGION Network 143: CPU01 Connection1 Status (Disabled)
   IF NOT #CPU01_CONN1_EN THEN
       #CPU01_CONN1_Send_St := INT#999;
       #CPU01_CONN1_Recv_St := INT#999;
   END_IF;
END_REGION

REGION Network 144: CPU00 Connection2 Status (Disabled)
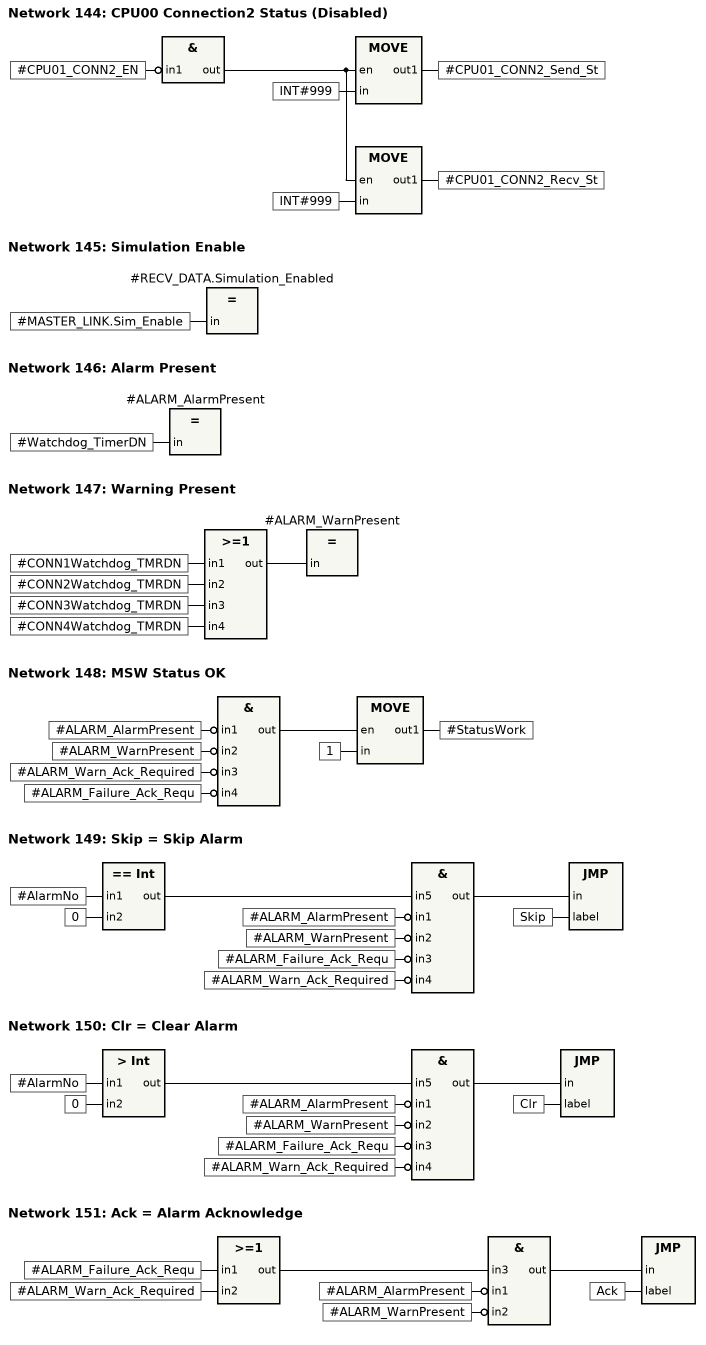
   IF NOT #CPU01_CONN2_EN THEN
       #CPU01_CONN2_Send_St := INT#999;
       #CPU01_CONN2_Recv_St := INT#999;
   END_IF;
END_REGION

REGION Network 145: Simulation Enable
   // >>>>>>>Simulation Enable>>>>>>>
   #RECV_DATA.Simulation_Enabled := #MASTER_LINK.Sim_Enable;
END_REGION

REGION Network 146: Alarm Present
   #ALARM_AlarmPresent := #Watchdog_TimerDN;
END_REGION

REGION Network 147: Warning Present
   #ALARM_WarnPresent := #CONN1Watchdog_TMRDN OR #CONN2Watchdog_TMRDN OR #CONN3Watchdog_TMRDN OR #CONN4Watchdog_TMRDN;
END_REGION

REGION Network 148: MSW Status OK
   IF NOT #ALARM_AlarmPresent AND NOT #ALARM_WarnPresent AND NOT #ALARM_Warn_Ack_Required AND NOT #ALARM_Failure_Ack_Requ THEN
       #StatusWork := 1;
   END_IF;
END_REGION

REGION Network 149: Skip = Skip Alarm
   // Skip = Skip Alarm
   IF (#AlarmNo = 0) AND NOT #ALARM_AlarmPresent AND NOT #ALARM_WarnPresent AND NOT #ALARM_Failure_Ack_Requ AND NOT #ALARM_Warn_Ack_Required THEN
       GOTO Skip;
   END_IF;
END_REGION

REGION Network 150: Clr = Clear Alarm
   // Clr = Clear Alarm
   IF (#AlarmNo > 0) AND NOT #ALARM_AlarmPresent AND NOT #ALARM_WarnPresent AND NOT #ALARM_Failure_Ack_Requ AND NOT #ALARM_Warn_Ack_Required THEN
       GOTO Clr;
   END_IF;
END_REGION

REGION Network 151: Ack = Alarm Acknowledge
   // Ack = Alarm Acknowledge
   IF (#ALARM_Failure_Ack_Requ OR #ALARM_Warn_Ack_Required) AND NOT #ALARM_AlarmPresent AND NOT #ALARM_WarnPresent THEN
       GOTO Ack;
   END_IF;
END_REGION

REGION Network 152: Communication Networks down
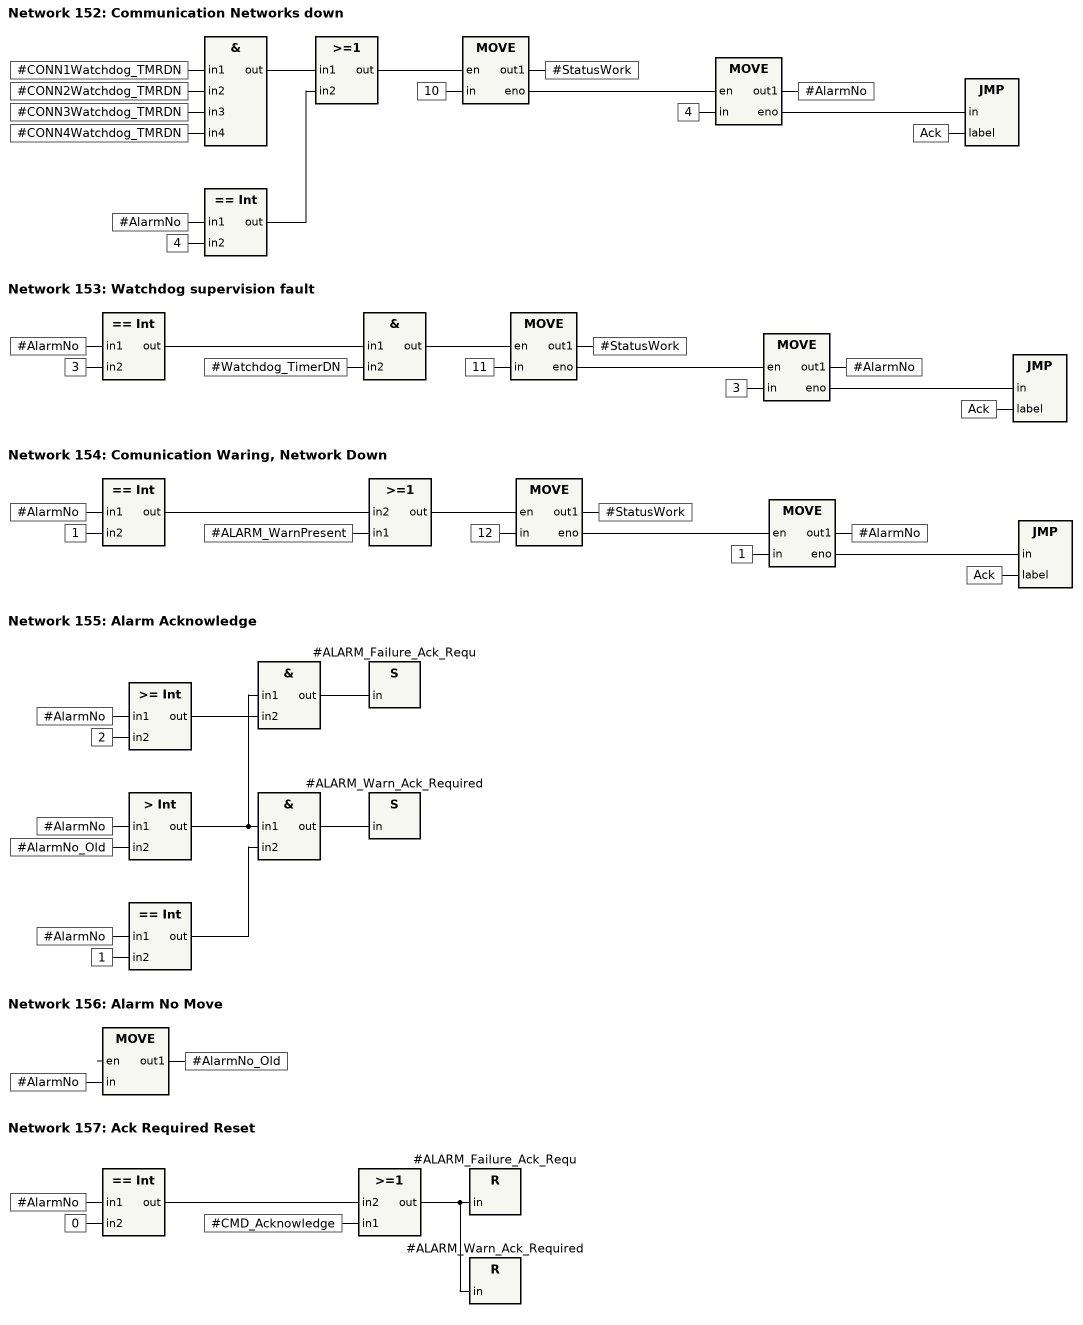
   // ENO of a box is taken as its EN; it also drops when the box reports an error
   #_w1 := (#CONN1Watchdog_TMRDN AND #CONN2Watchdog_TMRDN AND #CONN3Watchdog_TMRDN AND #CONN4Watchdog_TMRDN) OR (#AlarmNo = 4);
   IF #_w1 THEN
       #StatusWork := 10;
       #AlarmNo := 4;
       GOTO Ack;
   END_IF;
END_REGION

REGION Network 153: Watchdog supervision fault
   // ENO of a box is taken as its EN; it also drops when the box reports an error
   #_w1 := (#AlarmNo = 3) AND #Watchdog_TimerDN;
   IF #_w1 THEN
       #StatusWork := 11;
       #AlarmNo := 3;
       GOTO Ack;
   END_IF;
END_REGION

REGION Network 154: Comunication Waring, Network Down
   // ENO of a box is taken as its EN; it also drops when the box reports an error
   #_w1 := (#AlarmNo = 1) OR #ALARM_WarnPresent;
   IF #_w1 THEN
       #StatusWork := 12;
       #AlarmNo := 1;
       GOTO Ack;
   END_IF;
END_REGION

REGION Network 155: Alarm Acknowledge
   // >>>>>>>Alarm Acknowledge>>>>>>>
   Ack:
   #_w1 := #AlarmNo > #AlarmNo_Old;
   IF #_w1 AND (#AlarmNo >= 2) THEN #ALARM_Failure_Ack_Requ := TRUE; END_IF;
   IF #_w1 AND (#AlarmNo = 1) THEN #ALARM_Warn_Ack_Required := TRUE; END_IF;
END_REGION

REGION Network 156: Alarm No Move
   #AlarmNo_Old := #AlarmNo;
END_REGION

REGION Network 157: Ack Required Reset
   IF (#AlarmNo = 0) OR #CMD_Acknowledge THEN
       #ALARM_Failure_Ack_Requ := FALSE;
       #ALARM_Warn_Ack_Required := FALSE;
   END_IF;
END_REGION

REGION Network 158: Skip = Skip Alarm
   // Skip = Skip Alarm
